(* IEC 61131-3 sources: SCLTeamCoder/experiment/datasets/oscat/oscat_code (part 2) *)

(* ---- FACT.st ---- *)
FUNCTION FACT : DINT
VAR_INPUT
    X : INT;
END_VAR
IF X >= 0 AND X <= 12 THEN
	FACT := math.FACTS[X];
ELSE
	FACT := -1;
END_IF;

(* working code without array
IF X > 12 OR X < 0 THEN
	FACT := -1;
ELSIF X < 7 THEN
	FACT := 1;
	FOR i := 2 TO X DO
		FACT := FACT * i;
	END_FOR;
ELSE
	FACT := 5040;
	FOR i := 8 TO X DO
		FACT := FACT * i;
	END_FOR;
END_IF;
*)

(* revision history
hm 4.3.2007		rev 1.1
	changed a critical error where while loop was indefinite.

hm	10.12.2007	rev 1.2
	start value for i has changed to 2 for better performance

hm	10. mar 2008	rev 1.3
	changed output of fact to dint to allow bigger values

hm	27. oct. 2008	rev 1.4
	optimized code

hm	26. mar. 2011	rev 1.5
	using array math.facts
*)
END_FUNCTION

(* ---- FIB.st ---- *)
FUNCTION FIB : DINT
VAR_INPUT
    X : INT;
END_VAR

VAR
    t1 : DINT;
    t2 : DINT;
END_VAR
IF X < 0 OR X > 46 THEN
	FIB := -1;
ELSIF x < 2 THEN
	FIB := X;
	RETURN;
ELSE
	(* the fibonacci number is the sum of the two suceeding fibonaci numbers *)
	(* we store the numbers alternatively in t1 and t2 depending on pt *)
	t2 := 1;
	WHILE X > 3 DO
		X := X-2;
		t1 := t1 + t2;
		t2 := t1 + t2;
	END_WHILE;
	IF X > 2 THEN t1 := t1 + t2; END_IF;
	fib := t1 + t2;
END_IF;

(* alternative code for very big numbers

IF X < 31 THEN
	fib := 0.4472136 * (expn(1.618034,X) - expn(-0.618034,X));
ELSE
	fib := 0.4472133 * expn(1.618034,X);
END_IF;

*)

(* revision history
hm		27. dec 2007	rev 1.0
	original version

hm		2. jan 2008	rev 1.1
	deleted unused variable pt

hm		10. mar 2008	rev 1.2
	changed output to dint instead of real

hm		26. mar. 2008	rev 1.3
	function now returns -1 for input < 0 or > 46

*)
END_FUNCTION

(* ---- FILL.st ---- *)
FUNCTION FILL : string
VAR_INPUT
    C : BYTE;
    L : INT;
END_VAR

VAR
    i : INT;
    sx : STRING[1];
END_VAR
Sx := CHR_TO_STRING(c);
(* limit L to maximum 80 characters the length of a standard string *)
L := LIMIT(0,L,STRING_LENGTH);
(* create a string of characters to be connected to str *)
FOR i := 1 TO 8 DO
	FILL := CONCAT(FILL,FILL);
	IF L.7 THEN FILL := CONCAT(FILL,Sx); END_IF;
	L := SHL(L,1);
END_FOR;

(* revision histroy
hm	29. mar. 2008	rev 1.0
	original release

hm	17. dec. 2008	rev 1.1
	changed function chr to chr_to_string

*)
END_FUNCTION

(* ---- FIND_CHAR.st ---- *)
FUNCTION FIND_CHAR : INT
VAR_INPUT
    str : STRING(STRING_LENGTH);
    pos : INT;
END_VAR

VAR
    i : INT;
    pt : POINTER TO ARRAY [1..255] OF BYTE;
    stop : INT;
    X : BYTE;
END_VAR
pt := ADR(str);
stop := LEN(str);
FOR i := MAX(pos,1) TO stop DO;
	X := pt^[i];
	IF X > 31 AND ((setup.EXTENDED_ASCII AND X <> 127) OR (NOT setup.EXTENDED_ASCII AND X < 127)) THEN
		FIND_CHAR := i;
		RETURN;
	END_IF;
END_FOR;
FIND_CHAR := 0;

(* revision history
hm	29. feb 2008	rev 1.0
	original version

hm	26. mar. 2008	rev 1.1
	char will now accept extended ascii

hm	29. mar. 2008	rev 1.2
	changed STRING to STRING(STRING_LENGTH)

hm	21. oct. 2008	rev 1.3
	changes setup constants
	optimized code
*)
END_FUNCTION

(* ---- FIND_CTRL.st ---- *)
FUNCTION FIND_CTRL : INT
VAR_INPUT
    str : STRING(STRING_LENGTH);
    pos : INT;
END_VAR

VAR
    i : INT;
    pt : POINTER TO ARRAY[1..255] OF BYTE;
    stop : INT;
    x : BYTE;
END_VAR
pt := ADR(str);
stop := LEN(str);
FOR i := MAX(pos,1) TO stop DO;
	x := PT^[I];
	IF x < 32 OR X = 127 THEN
		FIND_CTRL := i;
		RETURN;
	END_IF;
END_FOR;
FIND_CTRL := 0;

(* revision history
hm	29. feb 2008	rev 1.0
	original version

hm	26. mar. 2008	rev 1.1
	character 127 is now recognized as control

hm	29. mar. 2008	rev 1.2
	changed STRING to STRING(STRING_LENGTH)
*)
END_FUNCTION

(* ---- FIND_NONUM.st ---- *)
FUNCTION FIND_NONUM : INT
VAR_INPUT
    str : STRING(STRING_LENGTH);
    pos : INT;
END_VAR

VAR
    i : INT;
    pt : POINTER TO ARRAY[1..255] OF BYTE;
    end : INT;
    X : BYTE;
END_VAR
pt := ADR(str);
end := LEN(str);
FOR i := MAX(pos,1) TO end DO;
	X := pt^[i];
	IF (X < 48 AND X <> 46) OR X > 57 THEN
		FIND_NONUM := i;
		RETURN;
	END_IF;
END_FOR;
FIND_NONUM := 0;

(* revision history
hm	6. oct. 2006	rev 1.0
	original version

hm	29. feb 2008	rev 1.1
	added input pos to start search at position

hm	29. mar. 2008	rev 1.2
	changed STRING to STRING(STRING_LENGTH)

hm	21. oct. 2008	rev 1.3
	optimized code

*)
END_FUNCTION

(* ---- FIND_NUM.st ---- *)
FUNCTION FIND_NUM : INT
VAR_INPUT
    str : STRING(SIZE := STRING_LENGTH);
    pos : INT;
END_VAR

VAR
    i : INT;
    pt : POINTER TO ARRAY[1..255] OF BYTE;
    stop : INT;
    X : BYTE;
END_VAR
pt := ADR(str);
stop := LEN(str);
FOR i := MAX(pos,1) TO stop DO;
	X := pt^[i];
	IF (X > 47 AND X < 58) OR X = 46 THEN
		FIND_NUM := i;
		RETURN;
	END_IF;
END_FOR;
FIND_NUM := 0;

(* revision history
hm	6. oct. 2006	rev 1.0
	original version

hm	29. feb 2008	rev 1.1
	added input pos to start search at position

hm	29. mar. 2008	rev 1.2
	changed STRING to STRING(STRING_LENGTH)

*)
END_FUNCTION

(* ---- FINDB.st ---- *)
FUNCTION FINDB : INT
VAR_INPUT
    str1 : STRING(STRING_LENGTH);
    str2 : STRING(STRING_LENGTH);
END_VAR

VAR
    pos : INT;
    length : INT;
END_VAR
length := LEN(str2);
FOR pos := LEN(str1) - length + 1 TO 1 BY -1 DO
	IF MID(str1,length,pos) = str2 THEN
		FindB := pos;
		RETURN;
	END_IF;
END_FOR;
FindB := 0;

(* revision history
hm	6. oct 2006		rev 1.0
	original version

hm	15 dec 2007		rev 1.1
	changed code for better performance

hm	29. feb 2008	rev 1.2
	added findb := 0 for compatibility reasons

hm	29. mar. 2008	rev 1.3
	changed STRING to STRING(STRING_LENGTH)
*)
END_FUNCTION

(* ---- FINDB_NONUM.st ---- *)
FUNCTION FINDB_NONUM : INT
VAR_INPUT
    str : STRING(STRING_LENGTH);
END_VAR

VAR
    pos : INT;
    pt : POINTER TO BYTE;
END_VAR
pt := ADR(str) + LEN(str) - 1;
FOR pos := LEN(str) TO 1 BY -1 DO;
	IF (PT^ < 48 AND PT^ <> 46) OR PT^ > 57 THEN
		FINDB_NONUM := pos;
		RETURN;
	END_IF;
	PT := PT - 1;
END_FOR;
FINDB_NONUM := 0;

(* revision history
hm	6. oct 2006		rev 1.0
	original version

hm	29. feb 2008	rev 1.1
	improved performance

hm	29. mar. 2008	rev 1.2
	changed STRING to STRING(STRING_LENGTH)

hm	21. oct. 2008	rev 1.3
	optimized code
*)
END_FUNCTION

(* ---- FINDB_NUM.st ---- *)
FUNCTION FINDB_NUM : INT
VAR_INPUT
    str : STRING:= STRING_LENGTH; // Input variable of type STRING with specified length
END_VAR

VAR
    pos : INT; // Local variable of type INT
    pt : POINTER TO BYTE; // Local variable of type pointer to BYTE
END_VAR
pt := ADR(str) + LEN(str) - 1;
FOR pos := LEN(str) TO 1 BY -1 DO;
	IF (PT^ > 47 AND PT^ < 58) OR PT^ = 46 THEN
		FINDB_NUM := pos;
		RETURN;
	END_IF;
	PT := PT - 1;
END_FOR;
FINDB_NUM := 0;

(* revision history
hm	6. oct 2006		rev 1.0
	original version

hm	29. feb 2008	rev 1.1
	improved performance

hm	29. mar. 2008	rev 1.2
	changed STRING to STRING(STRING_LENGTH)
*)
END_FUNCTION

(* ---- FINDP.st ---- *)
FUNCTION FINDP : INT
VAR_INPUT
    str : STRING[STRING_LENGTH];
    src : STRING[STRING_LENGTH];
    pos : INT;
END_VAR

VAR
    i : INT;
    ls : INT;
    lx : INT;
    stp : INT;
END_VAR
ls := LEN(str);
lx := LEN(src);
IF ls < lx OR lx = 0 THEN RETURN; END_IF;
stp := ls - lx + 1;
FOR i := MAX(pos,1) TO stp DO
	IF MID(str,lx,i) = src THEN
		FINDP := i;
		RETURN;
	END_IF;
END_FOR;
FINDP := 0;

(* revision histroy
hm	4. feb. 2008	rev 1.0
	original release

hm	29. feb 2008	rev 1.1
	ADDED MAX(pos,1) in loop initialization

hm	29. mar. 2008	rev 1.2
	changed STRING to STRING(STRING_LENGTH)
*)
END_FUNCTION

(* ---- FIX.st ---- *)
FUNCTION FIX : string
VAR_INPUT
    str : STRING[STRING_LENGTH];
    L : INT;
    C : BYTE;
    M : INT;
END_VAR

VAR
    N : INT;
    SX : STRING[STRING_LENGTH];
END_VAR
(* make sure L does not exceed the limits of a string *)
N := LIMIT(0,L,STRING_LENGTH) - LEN(str);
IF N <= 0 THEN
	(* truncate the string at length N *)
	IF M = 1 THEN
		FIX := RIGHT(str,L);
	ELSE
		FIX := LEFT(str,L);
	END_IF;
ELSIF M = 1 THEN
	(* connect fill characters at the beginning *)
	sx := FILL(C,N);
	FIX := CONCAT(sx,str);
ELSIF M = 2 THEN
	(* center str beween fill characters *)
	(* for an uneven number of fill characters, there is one more at the end *)
	sx := FILL(C,SHR(N+1,1));
	FIX := CONCAT(str,sx);
	SX := LEFT(sx,SHR(N,1));
	FIX := CONCAT(sx,FIX);
ELSE
	(* connect fill characters at the end *)
	SX := FILL(C,N);
	FIX := CONCAT(str,SX);
END_IF;

(* revision histroy
hm	29. mar. 2008	rev 1.0
	original release

*)
END_FUNCTION

(* ---- FLOAT_TO_REAL.st ---- *)
FUNCTION FLOAT_TO_REAL : REAL
VAR_INPUT
    FLT : STRING[20];
END_VAR

VAR
    pt : POINTER TO ARRAY[1..20] OF BYTE;
    i : INT;
    X : BYTE;
    sign : INT := 1;
    stop : INT;
    tmp : DINT;
    d : INT;
END_VAR
pt := ADR(FLT);
stop := LEN(FLT);

(* we first check for sign and exit if first number or dot is reached *)
FOR i := 1 TO stop DO
	X := pt^[i];
	IF X > 47 AND X < 58 OR X = 46 THEN
		EXIT;
	ELSIF X = 45 THEN
		(* code 45 is sign *)
		sign := -1;
	END_IF;
END_FOR;

(* now we scan numbers till end or dot or E is reached *)
FOR i := i TO stop DO
	X := pt^[i];
	IF X = 44 OR X = 46 OR X = 69 OR X = 101 THEN
		EXIT;
	(* calculate the value of the digit *)
	ELSIF X > 47 AND x < 58 THEN
		tmp := tmp * 10 + X - 48;
	END_IF;
END_FOR;

(* process the portion after the comma if comma or dot is reached exit if exponent starts *)
IF x = 44 OR X = 46 THEN
	FOR i := i + 1 TO stop DO
		X := pt^[i];
		IF X = 69 OR X = 101 THEN
			EXIT;
		ELSIF x > 47 AND x < 58 THEN
			tmp := tmp * 10 + X - 48;
			d := d - 1;
		END_IF;
	END_FOR;
END_IF;

(* process exponent if present *)
IF X = 69 OR X = 101 THEN
	d := d + DEC_TO_INT(RIGHT(FLT, stop - i));
END_IF;

FLOAT_TO_REAL :=  EXPN(10, d) * DINT_TO_REAL(TMP * SIGN);

(* revision histroy
hm	22. jun. 2008	rev 1.0
	original release

hm	2. oct. 2008	rev 1.1
	fixed an error, characters 8 and 9 would not be converted

hm	22. oct. 2008	rev 1.2
	last fix was not done correctly

hm	23. oct. 2008	rev 1.3
	optimzed code
*)
END_FUNCTION

(* ---- FLOOR.st ---- *)
FUNCTION FLOOR : INT
VAR_INPUT
    X : REAL;
END_VAR
FLOOR := REAL_TO_INT(X);
IF FLOOR > X THEN
	FLOOR := FLOOR - 1;
END_IF;

(* revision history
hm		7. feb 2007		rev 1.0
	originlal version

hm		21. mar. 2008	rev 1.1
	replaced trunc with real_to_int for compatibility reasons

*)
END_FUNCTION

(* ---- FLOOR2.st ---- *)
FUNCTION FLOOR2 : DINT
VAR_INPUT
    X : REAL;
END_VAR
FLOOR2 := REAL_TO_DINT(X);
IF DINT_TO_REAL(FLOOR2) > X THEN
	FLOOR2 := FLOOR2 - 1;
END_IF;

(* revision history
hm	21. mar. 2008	rev 1.0
	originlal version

hm	4. apr. 2008	rev 1.1
	added type conversion to avoid warnings under codesys 3.0
*)
END_FUNCTION

(* ---- FRACT.st ---- *)
FUNCTION FRACT : REAL
VAR_INPUT
    x : REAL;
END_VAR
IF ABS(x) < 2.0E9 THEN
	FRACT := x - DINT_TO_REAL(D_TRUNC(x));
ELSE
	FRACT := 0.0;
END_IF;

(* revision history
hm	4. aug 2006	rev 1.0
	original version

hm	11. mar 2008	rev 1.1
	added dint_to_real for compatibility reasons
	now returns 0 for number > 2e9
	changed input to x

hm	21. mar. 2008	rev 1.2
	use D_trunc instead of TRUNC for compatibility reasons

hm	10. mar. 2009	rev 1.3
	real constants updated to new systax using dot

*)
END_FUNCTION

(* ---- FRMP_B.st ---- *)
FUNCTION FRMP_B : BYTE
VAR_INPUT
    START : BYTE;
    DIR   : BOOL;
    TD    : TIME;
    TR    : TIME;
END_VAR
IF TD < TR THEN
	FRMP_B := MIN(DWORD_TO_BYTE(SHL(TIME_TO_DWORD(TD), 8) / TIME_TO_DWORD(TR)), SEL(DIR, START, BYTE#255 - START));
	IF DIR THEN
		FRMP_B := START + FRMP_B;
	ELSE
		FRMP_B := START - FRMP_B;
	END_IF;
ELSE
	FRMP_B := SEL(DIR, 0, 255);
END_IF;

(* revision history

17. feb. 2011	rev 1.0
	new module

*)
END_FUNCTION

(* ---- FSTRING_TO_BYTE.st ---- *)
FUNCTION FSTRING_TO_BYTE : BYTE
VAR_INPUT
    IN: STRING[12];
END_VAR
IF LEFT(IN, 2) = '2#' THEN
	(* we need to convert binary *)
	FSTRING_TO_BYTE := BIN_TO_BYTE(RIGHT(in, LEN(in) - 2));
ELSIF LEFT(in, 2) = '8#' THEN
	(* weneed to convert octals *)
	FSTRING_TO_BYTE := OCT_TO_BYTE(RIGHT(in, LEN(in) - 2));
ELSIF LEFT(in, 3) = '16#' THEN
	(* we need to convert hexadecimal *)
	FSTRING_TO_BYTE := HEX_TO_BYTE(RIGHT(in, LEN(in) - 3));
ELSE
	(* we assume decimal representation *)
	FSTRING_TO_BYTE := DEC_TO_BYTE(CLEAN(in,'0123456789'));
END_IF;

(* revision histroy
hm	18. jun. 2008	rev 1.0
	original release

hm	20. sep. 2008	rev 1.1
	changed length of input string from 20 to 12
*)
END_FUNCTION

(* ---- FSTRING_TO_DT.st ---- *)
FUNCTION FSTRING_TO_DT : DT
VAR_INPUT
    SDT: STRING[60];    // Input variable for source data text
    FMT: STRING[60];    // Input variable for format
END_VAR

VAR CONSTANT
    ignore: STRING[1] := '*';  // ignore character is *
    fchar: STRING[1] := '#';    // format character is #
END_VAR

VAR
    c: STRING[1];    // local variable for character
    tmp: STRING[20];  // local variable for temporary storage
    end: INT;         // local variable for end indicator
    dy: INT := 1970;  // local variable for year, initialized to 1970
    dm: INT := 1;     // local variable for month, initialized to 1
    dd: INT := 1;     // local variable for day, initialized to 1
    th: INT;         // local variable for hour
    tm: INT;         // local variable for minute
    ts: INT;         // local variable for second
END_VAR
(* scan input string *)
WHILE fmt <> '' DO
	c := LEFT(fmt,1);
	IF c = ignore THEN
		(* skip ignore characters *)
		fmt := DELETE(fmt,1,1);
		sdt := DELETE(sdt,1,1);
	ELSIF C = fchar THEN
		(* format chracter found skip format char and read identifier *)
		(* store format identifier in c and skip to next char in fmt *)
		c := MID(fmt,1,2);
		fmt := DELETE(fmt,2,1);
		(* extract the substring until the end of sdt or to next char of fmt *)
		IF fmt = '' THEN
			tmp := sdt;
		ELSE
			(* serach for end of substring *)
			end := FIND(sdt, LEFT(fmt,1))-1;
			tmp := LEFT(sdt, end);
			sdt := DELETE(sdt, end,1);
		END_IF;
		(* extract information from substring *)
		IF c = 'Y' THEN
			dy := STRING_TO_INT(tmp);
			IF dy < 100 THEN dy := dy + 2000; END_IF;
		ELSIF c = 'M' THEN
			dm := STRING_TO_INT(tmp);
		ELSIF c = 'N' THEN
			dm := FSTRING_TO_MONTH(tmp,0);
		ELSIF c = 'D' THEN
			dd := STRING_TO_INT(tmp);
		ELSIF c = 'h' THEN
			th := STRING_TO_INT(tmp);
		ELSIF c = 'm' THEN
			tm := STRING_TO_INT(tmp);
		ELSIF c = 's' THEN
			ts := STRING_TO_INT(tmp);
		END_IF;
	ELSIF c = LEFT(sdt,1) THEN
		(* skip matching characters *)
		fmt := DELETE(fmt,1,1);
		sdt := DELETE(sdt,1,1);
	ELSE
		RETURN;
	END_IF;
END_WHILE;

FSTRING_TO_DT := SET_DT(dy,dm,dd,th,tm,ts);

(* revision histroy
hm	24. sep. 2008	rev 1.0
	original release

*)
END_FUNCTION

(* ---- FSTRING_TO_DWORD.st ---- *)
FUNCTION FSTRING_TO_DWORD : DWORD
VAR_INPUT
    IN : STRING[40];
END_VAR
IF LEFT(IN, 2) = '2#' THEN
	(* we need to convert binary *)
	FSTRING_TO_DWORD := BIN_TO_DWORD(RIGHT(in, LEN(in) - 2));
ELSIF LEFT(in, 2) = '8#' THEN
	(* weneed to convert octals *)
	FSTRING_TO_DWORD := OCT_TO_DWORD(RIGHT(in, LEN(in) - 2));
ELSIF LEFT(in, 3) = '16#' THEN
	(* we need to convert hexadecimal *)
	FSTRING_TO_DWORD := HEX_TO_DWORD(RIGHT(in, LEN(in) - 3));
ELSE
	(* we assume decimal representation *)
	FSTRING_TO_DWORD := DEC_TO_DWORD(CLEAN(in,'0123456789'));
END_IF;

(* revision histroy
hm	18. jun. 2008	rev 1.0
	original release

hm	20. sep. 2008	rev 1.1
	changed length of input dtring from 20 to 40

*)
END_FUNCTION

(* ---- FSTRING_TO_MONTH.st ---- *)
FUNCTION FSTRING_TO_MONTH : INT
VAR_INPUT
    MTH : STRING(20);
    LANG : INT;
END_VAR

VAR
    lx : INT;
END_VAR
IF LANG = 0 THEN lx := LANGUAGE.DEFAULT; ELSE lx := MIN(LANG, LANGUAGE.LMAX); END_IF;
MTH := TRIM(mth);
MTH := CAPITALIZE(LOWERCASE(MTH));

FOR FSTRING_TO_MONTH := 1 TO 12 DO
	IF MTH = language.MONTHS[lx, FSTRING_TO_MONTH] THEN RETURN; END_IF;
	IF MTH = language.MONTHS3[lx, FSTRING_TO_MONTH] THEN RETURN; END_IF;
END_FOR;

(* since no name matched try to decode as integer *)
FSTRING_TO_MONTH := STRING_TO_INT(MTH);

(* revision histroy
hm	25. sep. 2008	rev 1.0
	original release

hm	19. oct. 2008	rev 1.1
	changed language setup constants

hm	25. oct. 2008	rev 1.2
	optimized code
*)
END_FUNCTION

(* ---- FSTRING_TO_WEEK.st ---- *)
FUNCTION FSTRING_TO_WEEK : BYTE
VAR_INPUT
    WEEK : STRING[60];
    LANG : INT;
END_VAR

VAR
    pos : INT;
END_VAR
pos := FIND(WEEK, ',');
WHILE pos > 0 DO
	FSTRING_TO_WEEK := FSTRING_TO_WEEK OR SHR(BYTE#128, FSTRING_TO_WEEKDAY(MID(WEEK, pos - 1, 1), LANG));
	WEEK := RIGHT(WEEK, LEN(Week) - pos);
	pos := FIND(WEEK, ',');
END_WHILE;
FSTRING_TO_WEEK := (FSTRING_TO_WEEK OR SHR(BYTE#128, FSTRING_TO_WEEKDAY(WEEK, LANG))) AND BYTE#127;

(* revision histroy
hm	18. jun. 2008	rev 1.0
	original release

hm	25. oct. 2008	rev 1.1
	using language defauls and input lang
*)
END_FUNCTION

(* ---- FSTRING_TO_WEEKDAY.st ---- *)
FUNCTION FSTRING_TO_WEEKDAY : INT
VAR_INPUT
    WDAY : STRING[20];
    LANG : INT;
END_VAR

VAR
    tmp : STRING[2];
    i : INT;
    ly : INT;
END_VAR
IF LANG = 0 THEN ly := LANGUAGE.DEFAULT; ELSE ly := MIN(LANG, LANGUAGE.LMAX); END_IF;
(* tmp needs to be calculated first otherwise find can return wrong values *)
tmp := TRIM(wday);
tmp := CAPITALIZE(LOWERCASE(tmp));
FOR i := 1 TO 7 DO
	IF language.WEEKDAYS2[ly, i] = tmp THEN
		FSTRING_TO_WEEKDAY := i;
		RETURN;
	END_IF;
END_FOR;
FSTRING_TO_WEEKDAY := STRING_TO_INT(WDAY);

(* revision histroy
hm	18. jun. 2008	rev 1.0
	original release

hm	18. jul. 2008	rev 1.1
	changed nested call of left(trim()) for compatibility reasons

hm	25. oct. 2008	rev 1.2
	using language constants
*)
END_FUNCTION

(* ---- GAMMA.st ---- *)
FUNCTION GAMMA : REAL
VAR_INPUT
    X : REAL;
END_VAR
IF x > 0.0 THEN
	GAMMA := SQRT(math.PI2 / X) * EXPT(math.E_INV * (x + 1.0 / (12.0 * x - 0.1 / X)), X);
END_IF;

(* the stirling formula is not very accurate for small values of X
IF X >=0 THEN GAMMA := SQRT(math.PI2 * X) * EXPT(X / math.E, X); END_IF;
*)

(* revision history
hm	10.12.2007	rev 1.0
	original version

hm	18. oct. 2008	rev 1.1
	using math constants

hm	26. oct. 2008	rev 1.2
	using new formula with better accuracy

hm	10. mar. 2009	rev 1.3
	real constants updated to new systax using dot

*)
END_FUNCTION

(* ---- GAUSS.st ---- *)
FUNCTION GAUSS : REAL
VAR_INPUT
    X : REAL;
    U : REAL;
    SI : REAL;
END_VAR

VAR
    temp : REAL;
    si_inv : REAL;
END_VAR
temp := X - U;
si_inv := 1.0  / si;
GAUSS := EXP(Temp * Temp * si_inv * si_inv * - 0.5) * 0.39894228 * si_inv;

(* revision hisdtory
hm	6. apr. 2008	rev 1.0
	original version

hm	27. oct. 2008	rev 1.1
	optimized performance

hm	10. mar. 2009	rev 1.2
	real constants updated to new systax using dot

*)
END_FUNCTION

(* ---- GAUSSCD.st ---- *)
FUNCTION GAUSSCD : REAL
VAR_INPUT
    X : REAL;
    U : REAL;
    SI : REAL;
END_VAR
GAUSSCD := (ERF((X - U) / (SI * 1.414213562)) + 1.0) * 0.5;

(* revision hisdtory
hm	6. apr. 2008	rev 1.0
	original version

hm	10. mar. 2009	rev 1.1
	real constants updated to new systax using dot

*)
END_FUNCTION

(* ---- GCD.st ---- *)
FUNCTION GCD : INT
VAR_INPUT
    A : DINT;
    B : DINT;
END_VAR

VAR
    t : DINT;
END_VAR
IF A = 0 THEN
	GCD := DINT_TO_INT(ABS(B));
ELSIF B = 0 THEN
	GCD := DINT_TO_INT(ABS(A));
ELSE
	A := ABS(A);
	B := ABS(B);
	GCD := 1;
	WHILE NOT(A.0 OR B.0) DO
		A := SHR(A,1);
		B := SHR(B,1);
		GCD := SHL(GCD,1);
	END_WHILE;
	WHILE A > 0 DO
		IF NOT(A.0) THEN A := SHR(A,1);
		ELSIF NOT(B.0) THEN B := SHR(B,1);
		ELSE
			t:= SHR(ABS(A-B),1);
			IF A < B THEN B := t; ELSE A := T; END_IF;
		END_IF;
	END_WHILE;
	GCD := GCD * DINT_TO_INT(B);
END_IF;

(* revision history
hm	19. jan. 2011	rev 1.0
	original version

*)
END_FUNCTION

(* ---- GDF.st ---- *)
FUNCTION GDF : REAL
VAR_INPUT
    X : REAL;
END_VAR
IF X = 0.0 THEN
	GDF := 0.0;
ELSIF X > 15.0 THEN
	GDF := math.PI05;
ELSIF X < -15.0 THEN
	GDF := -math.PI05;
ELSE
	GDF := ATAN(EXP(X)) * 2.0 - math.PI05;
END_IF;

(* revision history
hm	27. apr. 2008	rev 1.0
	original version

hm	18. oct. 2008	rev 1.1
	using math constants

hm	10. mar. 2009	rev 1.2
	real constants updated to new systax using dot

*)
END_FUNCTION

(* ---- GEO_TO_DEG.st ---- *)
FUNCTION GEO_TO_DEG : REAL
VAR_INPUT
    D : INT;
    M : INT;
    SEC : REAL;
END_VAR
GEO_TO_DEG := INT_TO_REAL(D) + INT_TO_REAL(M) * 0.016666666666667 + sec * 0.00027777777777778;

(* revision histroy
hm	22. jan. 2009	rev 1.0
	original release

*)
END_FUNCTION

(* ---- GOLD.st ---- *)
FUNCTION GOLD : REAL
VAR_INPUT
    X : REAL;
END_VAR
GOLD := (X + SQRT(X*X + 4.0)) * 0.5;

(* revision history
hm	27. apr. 2008	rev 1.0
	original version

hm	10. mar. 2009	rev 1.1
	real constants updated to new systax using dot

*)
END_FUNCTION

(* ---- GRAY_TO_BYTE.st ---- *)
FUNCTION GRAY_TO_BYTE : BYTE
VAR_INPUT
    IN : BYTE;
END_VAR
GRAY_TO_BYTE := SHR(IN,4) XOR IN;
GRAY_TO_BYTE := SHR(GRAY_TO_BYTE,2) XOR GRAY_TO_BYTE;
GRAY_TO_BYTE := SHR(GRAY_TO_BYTE,1) XOR GRAY_TO_BYTE;

(* revision history
hm	9. nov. 2009	rev 1.0
	original version

*)
END_FUNCTION

(* ---- HEX_TO_BYTE.st ---- *)
FUNCTION HEX_TO_BYTE : BYTE
VAR_INPUT
    HEX : STRING(5);
END_VAR

VAR
    pt : POINTER TO BYTE;
    i : INT;
    X : BYTE;
    stop : INT;
END_VAR
pt := ADR(hex);
stop := LEN(hex);
FOR I := 1 TO stop DO
	(* read the first character and subtract 48 to get value in decimal 0 = 48 *)
	x := pt^;
	(* calculate the value of the digit *)
	IF X > 47 AND x < 58 THEN
		HEX_TO_BYTE := SHL(HEX_TO_BYTE,4) + X - 48;
	ELSIF X > 64 AND X < 71 THEN
		HEX_TO_BYTE := SHL(HEX_TO_BYTE,4) + X - 55;
	ELSIF X > 96 AND X < 103 THEN
		HEX_TO_BYTE := SHL(HEX_TO_BYTE,4) + X - 87;
	END_IF;
	pt := pt + 1;
END_FOR;

(* revision histroy
hm	18. jun. 2008	rev 1.0
	original release

hm	20. sep.2008	rev 1.1
	changed length of input string from 20 to 5

*)
END_FUNCTION

(* ---- HEX_TO_DWORD.st ---- *)
FUNCTION HEX_TO_DWORD : DWORD
VAR_INPUT
    Hex: STRING[20];
END_VAR

VAR
    pt: POINTER TO BYTE;
    i: INT;
    X: BYTE;
    stop: INT;
END_VAR
pt := ADR(hex);
stop := LEN(hex);
FOR I := 1 TO stop DO
	(* read the first character and subtract 48 to get value in decimal 0 = 48 *)
	x := pt^;
	(* calculate the value of the digit *)
	IF X > 47 AND x < 58 THEN
		HEX_TO_DWORD := SHL(HEX_TO_DWORD,4) + X - 48;
	ELSIF X > 64 AND X < 71 THEN
		HEX_TO_DWORD := SHL(HEX_TO_DWORD,4) + X - 55;
	ELSIF X > 96 AND X < 103 THEN
		HEX_TO_DWORD := SHL(HEX_TO_DWORD,4) + X - 87;
	END_IF;
	pt := pt + 1;
END_FOR;

(* revision histroy
hm	2.10.2007		rev 1.0
	original release

hm	19.11.2007		rev 1.1
	changed type of function from int to dword

hm 	4. mar 2008		rev 1.2
	added support for a..f and return 0 for invalid string

hm	29. mar. 2008	rev 1.3
	changed STRING to STRING(8)

hm	18. jun. 2008	rev 1.4
	changed input hex to STRING(20)
	function now ignores wrong characters
*)
END_FUNCTION

(* ---- HOUR.st ---- *)
FUNCTION HOUR : INT
VAR_INPUT
    itod : TIME_OF_DAY; // Declaration of input variable itod of type TIME_OF_DAY
END_VAR
HOUR := DWORD_TO_INT(TOD_TO_DWORD(itod) / 3600000);

(* change history
hm 4. aug 2006	rev 1.0
	original version

hm 2.10.2006 	rev 1.1
	changed name of input to itod

*)
END_FUNCTION

(* ---- HOUR_OF_DT.st ---- *)
FUNCTION HOUR_OF_DT : INT
VAR_INPUT
    XDT : DT;
END_VAR
HOUR_OF_DT := DWORD_TO_INT((DT_TO_DWORD(XDT) MOD 86400) / 3600);

(* revision history
hm		6.9.2008	rev 1.0
	original version

*)
END_FUNCTION

(* ---- HOUR_TO_TIME.st ---- *)
FUNCTION HOUR_TO_TIME : TIME
VAR_INPUT
    IN : REAL;
END_VAR
HOUR_TO_TIME := DWORD_TO_TIME(REAL_TO_DWORD(IN * 3600000));

(* revision history
hm		4. aug 2006	rev 1.0
	original version

hm	14. mar. 2008	rev 1.1
	rounded the input after the last digit

hm	24. feb. 2009	rev 1.2
	changed input to IN
*)
END_FUNCTION

(* ---- HOUR_TO_TOD.st ---- *)
FUNCTION HOUR_TO_TOD : TOD
VAR_INPUT
    IN : REAL;
END_VAR
HOUR_TO_TOD := DWORD_TO_TOD(REAL_TO_DWORD(IN * 3600000));

(* revision history
hm	4. aug. 2006	rev 1.0
	original version

hm	14. mar. 2008	rev 1.1
	rounded the input after the last digit

hm	24. feb. 2009	rev 1.2
	changed input to IN
*)
END_FUNCTION

(* ---- HYPOT.st ---- *)
FUNCTION HYPOT : REAL
VAR_INPUT
    X : REAL;
    Y : REAL;
END_VAR
HYPOT := SQRT(x*x + y*y);

(* revision history
hm	21. feb 2008	rev 1.0
	original version

*)
END_FUNCTION

(* ---- INC.st ---- *)
FUNCTION INC : INT
VAR_INPUT
    X : INT;
    D : INT;
    M : INT;
END_VAR
INC := (X + D + M + 1) MOD (M + 1);

(* revision history
hm	7. feb 2007		REV 1.0
	original version

hm	15. jan 2008	rev 1.1
	allow for neagtive increment

*)
END_FUNCTION

(* ---- INC1.st ---- *)
FUNCTION INC1 : INT
VAR_INPUT
    X : INT;
    N : INT;
END_VAR
IF X >= N - 1 THEN
	INC1 := 0;
ELSE
	INC1 := X + 1;
END_IF;

(* revision history
hm	13. oct. 2008	rev 1.0
	original version

hm	22. oct. 2008	rev 1.1
	added statement to return value for compatibility reasons

hm	23. feb. 2009	rev 1.2
 	when inc1 is called with X >= N inc will continue with 0
*)
END_FUNCTION

(* ---- INC2.st ---- *)
FUNCTION INC2 : INT
VAR_INPUT
    X : INT;
    D : INT;
    L : INT;
    U : INT;
END_VAR

VAR
    tmp : INT;
END_VAR
tmp := U - L + 1;
INC2 := (X + D - L + tmp) MOD tmp + L;

(* revision history
hm	29. jun. 2008		REV 1.0
	original version

*)
END_FUNCTION

(* ---- INT_TO_BCDC.st ---- *)
FUNCTION INT_TO_BCDC : BYTE
VAR_INPUT
    IN : INT;
END_VAR
INT_TO_BCDC := SHL(INT_TO_BYTE(IN / INT#10),4) OR INT_TO_BYTE(in MOD INT#10);

(* revision history
hm	13.12.2007
	original version

hm	30.6.2008	rev 1.1
	changed name INT_TO_BCD to INT_TO_BCDC to avoid collision with util.lib
	corrected error in code

*)
END_FUNCTION

(* ---- INV.st ---- *)
FUNCTION INV : REAL
VAR_INPUT
    X : REAL;
END_VAR
IF X <> 0.0 THEN INV := 1.0 / X; END_IF;

(* revision history
hm	26. oct. 2008	rev 1.0
	original version

hm	10. mar. 2009	rev 1.1
	real constants updated to new systax using dot

*)
END_FUNCTION

(* ---- IS_ALNUM.st ---- *)
FUNCTION IS_ALNUM : BOOL
VAR_INPUT
    str : STRING(STRING_LENGTH);
END_VAR_INPUT

VAR
    L : INT;
    pt : POINTER TO BYTE;
    pos : INT;
END_VAR
PT := ADR(str);
L := LEN(str);
FOR pos := 1 TO L DO
	IF NOT (ISC_ALPHA(pt^) OR ISC_NUM(pt^)) THEN
		IS_ALNUM := FALSE;
		RETURN;
	END_IF;
    	PT := PT + 1;
END_FOR;
IS_ALNUM := L > 0;

(* revision history
hm	29. feb 2008	rev 1.0
	original version

hm	29. mar. 2008	rev 1.1
	changed STRING to STRING(STRING_LENGTH)
*)
END_FUNCTION

(* ---- IS_ALPHA.st ---- *)
FUNCTION IS_ALPHA : BOOL
VAR_INPUT
    str: STRING(STRING_LENGTH);
END_VAR

VAR
    L: INT;
    pt: POINTER TO BYTE;
    pos: INT;
END_VAR
PT := ADR(str);
L := LEN(str);
FOR pos := 1 TO L DO
	IF NOT ISC_ALPHA(pt^) THEN
		IS_ALPHA := FALSE;
		RETURN;
	END_IF;
    	PT := PT + 1;
END_FOR;
IS_ALPHA := L > 0;

(* revision history
hm	29. feb 2008	rev 1.0
	original version

hm	29. mar. 2008	rev 1.1
	changed STRING to STRING(STRING_LENGTH)
*)
END_FUNCTION

(* ---- IS_CC.st ---- *)
FUNCTION IS_CC : BOOL
VAR_INPUT
    str : STRING(STRING_LENGTH);
    cmp : STRING(STRING_LENGTH);
END_VAR

VAR
    L : INT;
    pos : INT;
END_VAR
L := LEN(str);
FOR pos := 1 TO L DO
	IF FIND(CMP,MID(str,1,pos)) = 0 THEN RETURN; END_IF;
END_FOR;
IS_CC := L > 0;

(* revision history
hm	19. mar 2008	rev 1.0
	original version

hm	29. mar. 2008	rev 1.1
	changed STRING to STRING(STRING_LENGTH)
*)
END_FUNCTION

(* ---- IS_CTRL.st ---- *)
FUNCTION IS_CTRL : BOOL
VAR_INPUT
    STR : STRING(STRING_LENGTH);
END_VAR

VAR
    L : INT;
    pt : POINTER TO BYTE;
    pos : INT;
END_VAR
PT := ADR(str);
L := LEN(str);
FOR pos := 1 TO L DO
	IF NOT (ISC_CTRL(pt^)) THEN
		IS_CTRL := FALSE;
		RETURN;
	END_IF;
    	PT := PT + 1;
END_FOR;
IS_CTRL := L > 0;

(* revision history
hm	29. feb. 2008	rev 1.0
	original version

hm	29. mar. 2008	rev 1.1
	changed STRING to STRING(STRING_LENGTH)
*)
END_FUNCTION

(* ---- IS_HEX.st ---- *)
FUNCTION IS_HEX : BOOL
VAR_INPUT
    str : STRING[STRING_LENGTH];
END_VAR

VAR
    L : INT;
    pt : POINTER TO BYTE;
    pos : INT;
END_VAR
PT := ADR(str);
L := LEN(str);
FOR pos := 1 TO L DO
	IF NOT (ISC_HEX(pt^)) THEN
		IS_HEX := FALSE;
		RETURN;
	END_IF;
    	PT := PT + 1;
END_FOR;
IS_HEX := L > 0;

(* revision history
hm	29. feb 2008	rev 1.0
	original version

hm	29. mar. 2008	rev 1.1
	changed STRING to STRING(STRING_LENGTH)
*)
END_FUNCTION

(* ---- IS_LOWER.st ---- *)
FUNCTION IS_LOWER : BOOL
VAR_INPUT
    str : STRING[STRING_LENGTH]; // Input variable declaration
END_VAR

VAR
    l : INT; // Local variable declaration
    pt : POINTER TO BYTE; // Pointer variable declaration
    pos : INT; // Position variable declaration
END_VAR
PT := ADR(str);
L := LEN(str);
FOR pos := 1 TO L DO
	IF NOT (ISC_LOWER(pt^)) THEN
		IS_LOWER := FALSE;
		RETURN;
	END_IF;
    	PT := PT + 1;
END_FOR;
IS_LOWER := L > 0;

(* revision history
hm	29. feb 2008	rev 1.0
	original version

hm	29. mar. 2008	rev 1.1
	changed STRING to STRING(STRING_LENGTH)
*)
END_FUNCTION

(* ---- IS_NCC.st ---- *)
FUNCTION IS_NCC : BOOL
VAR_INPUT
    str : STRING[STRING_LENGTH];
    cmp : STRING[STRING_LENGTH];
END_VAR

VAR
    L : INT;
    pos : INT;
END_VAR
L := LEN(str);
FOR pos := 1 TO L DO
	IF FIND(CMP,MID(str,1,pos)) > 0 THEN RETURN; END_IF;
END_FOR;
IS_NCC := TRUE;

(* revision history
hm	19. mar 2008	rev 1.0
	original version

hm	29. mar. 2008	rev 1.1
	changed STRING to STRING(STRING_LENGTH)
*)
END_FUNCTION

(* ---- IS_NUM.st ---- *)
FUNCTION IS_NUM : BOOL
VAR_INPUT
    str : STRING[STRING_LENGTH];  // Input variable of type STRING with specified length
END_VAR

VAR
    L : INT;                       // Local variable of type INT
    pt : POINTER TO BYTE;         // Local variable, pointer to BYTE
    pos : INT;                    // Local variable of type INT
END_VAR
PT := ADR(str);
L := LEN(str);
FOR pos := 1 TO L DO
	IF NOT (ISC_NUM(pt^)) THEN
		IS_NUM := FALSE;
		RETURN;
	END_IF;
    	PT := PT + 1;
END_FOR;
IS_NUM := L > 0;

(* revision history
hm	29. feb 2008	rev 1.0
	original version

hm	29. mar. 2008	rev 1.1
	changed STRING to STRING(STRING_LENGTH)
*)
END_FUNCTION

(* ---- IS_SORTED.st ---- *)
FUNCTION IS_SORTED : BOOL
VAR_INPUT
    pt : ^ ARRAY [0..32000] OF REAL; // Pointer to an array of REAL
    size : UINT; // Size variable of type UINT
END_VAR

VAR
    stop : INT; // Local variable of type INT
    i : INT; // Local variable of type INT
END_VAR
stop := UINT_TO_INT(SHR(size,2)-2);
FOR i := 0 TO stop DO
	IF pt^[i] > pt^[i+1] THEN
		IS_SORTED := FALSE;
		RETURN;
	END_IF;
END_FOR;

IS_SORTED := TRUE;

(* revision history

hm 	29. mar. 2008 	rev 1.0
	original version

hm	4. apr. 2008	rev 1.1
	added type conversion to avoid warnings under codesys 3.0
*)
END_FUNCTION

(* ---- IS_UPPER.st ---- *)
FUNCTION IS_UPPER : BOOL
VAR_INPUT
    str : STRING; // Length to be defined as per application requirements
END_VAR

VAR
    L : INT;
    pt : POINTER TO BYTE;
    pos : INT;
END_VAR
PT := ADR(str);
L := LEN(str);
FOR pos := 1 TO L DO
	IF NOT (ISC_UPPER(pt^)) THEN
		IS_UPPER := FALSE;
		RETURN;
	END_IF;
    	PT := PT + 1;
END_FOR;
IS_UPPER := L > 0;

(* revision history
hm	29. feb 2008	rev 1.0
	original version

hm	29. mar. 2008	rev 1.1
	changed STRING to STRING(STRING_LENGTH)
*)
END_FUNCTION

(* ---- ISC_ALPHA.st ---- *)
FUNCTION ISC_ALPHA : BOOL
#VAR_INPUT
    IN : BYTE;
END_VAR
IF setup.EXTENDED_ASCII THEN
	ISC_ALPHA := (in > 64 AND in < 91) OR (in > 191  AND in <> 215 AND in <> 247) OR (in > 96 AND in < 123);
ELSE
	ISC_ALPHA := (IN > 64 AND IN < 91) OR (in > 96 AND in < 123);
END_IF;

(* revision history
hm	6. mar. 2008	rev 1.0
	original version

hm	19. oct. 2008	rev 1.1
	changes setup constants
*)
END_FUNCTION

(* ---- ISC_CTRL.st ---- *)
FUNCTION ISC_CTRL : BOOL
VAR_INPUT
    IN : BYTE;
END_VAR
ISC_CTRL := IN < 32 OR IN = 127;

(* revision history
hm		6. mar. 2008	rev 1.0
	original version

*)
END_FUNCTION

(* ---- ISC_HEX.st ---- *)
FUNCTION ISC_HEX : BOOL
VAR_INPUT
    IN : BYTE;
END_VAR
ISC_HEX := (IN > 47 AND IN < 58) OR (IN > 64 AND IN < 71) OR (IN > 96 AND IN < 103);

(* revision history
hm		6. mar. 2008	rev 1.0
	original version

*)
END_FUNCTION

(* ---- ISC_LOWER.st ---- *)
FUNCTION ISC_LOWER : BOOL
VAR_INPUT
    IN : BYTE; // Input variable
END_VAR
IF setup.EXTENDED_ASCII THEN
	ISC_LOWER := ((in > 96) AND (in < 123)) OR ((in > 222) AND (in <> 247));
ELSE
	ISC_LOWER := ((in > 96) AND (in < 123));
END_IF;

(* revision history
hm	6. mar. 2008	rev 1.0
	original version

hm	19. oct. 2008	rev 1.1
	changes setup constants
*)
END_FUNCTION

(* ---- ISC_NUM.st ---- *)
FUNCTION ISC_NUM : BOOL
VAR_INPUT
    IN : BYTE;
END_VAR
ISC_NUM := IN > 47 AND IN < 58;

(* revision history
hm		6. mar. 2008	rev 1.0
	original version

*)
END_FUNCTION

(* ---- ISC_UPPER.st ---- *)
FUNCTION ISC_UPPER : BOOL
VAR_INPUT
    IN : BYTE;
END_VAR
IF setup.EXTENDED_ASCII THEN
	ISC_UPPER :=  ((in > 64) AND (in < 91)) OR (((in > 191) AND (in < 223)) AND (in <> 215));
ELSE
	ISC_UPPER := ((in > 64) AND (in < 91));
END_IF;

(* revision history
hm	6. mar. 2008	rev 1.0
	original version

hm	19. oct. 2008	rev 1.1
	changes setup constants

*)
END_FUNCTION

(* ---- JD2000.st ---- *)
FUNCTION JD2000 : REAL
VAR_INPUT
    DTI : TIME;
END_VAR
JD2000 := DWORD_TO_REAL(DT_TO_DWORD(DTI) - 946728000) / 86400.0;

(* revision histroy
hm	15. jul. 2008	rev 1.0
	original release

*)
END_FUNCTION

(* ---- K_TO_C.st ---- *)
FUNCTION K_TO_C : REAL
VAR_INPUT
    Kelvin : REAL;
END_VAR
K_TO_C := Kelvin + phys.T0;

(* revision history

hm	4. aug 2006	rev 1.0
	original version

hm	19. aug 2009	rev 1.1
	fixed calculation error

*)
END_FUNCTION

(* ---- KMH_TO_MS.st ---- *)
FUNCTION KMH_TO_MS : REAL
VAR_INPUT
    kmh : REAL;
END_VAR
KMH_TO_MS := kmh * 0.2777777777777;

(* revision history
hm	4. feb 2007		rev 1.0
	original version

hm	6. jan 2008		rev 1.1
	improved performance

*)
END_FUNCTION

(* ---- LAMBERT_W.st ---- *)
FUNCTION LAMBERT_W : REAL
VAR_INPUT
    X : REAL;
END_VAR

VAR
    w : REAL;
    i : INT;
    we : REAL;
    w1e : REAL;
    last : DWORD;
    ewx : REAL;
END_VAR
(* check for valid input and return -1000 if too low *)
IF x < -0.367879441171442 THEN
	LAMBERT_W := -1000.0;
	RETURN;
(* return 0 if x = 0 *)
ELSIF x = 0.0 THEN
	RETURN;
(* first an estimate is calculated *)
ELSIF x <= 500.0 THEN
	w := LN(x + 1.0);
	w := 0.665 * (1.0 + 0.0195 * w) * w + 0.04;
ELSE
	w := LN(x - 4.0) - (1.0 - 1.0/LN(x)) * LN(LN(x));
END_IF;
(* use estimate to calculate exact result *)
FOR i := 0 TO 5 DO
	ewx := EXP(w);
	we := w * ewx - x;
	w1e := (w+1.0) * ewx;
	last := REAL_TO_DW(w) AND 16#FFFF_FFFC;
	w := w - (we / (w1e - (w+2.0) * we / (2.0 * w + 2.0)));
	IF (REAL_TO_DW(w) AND 16#FFFF_FFFC) = last THEN EXIT; END_IF;
END_FOR;
LAMBERT_W := w;

(* revision hisdtory
hm	26. oct. 2008	rev 1.0
	original version

hm	10. mar. 2009	rev 1.1
	real constants updated to new systax using dot

*)
END_FUNCTION

(* ---- LANGEVIN.st ---- *)
FUNCTION LANGEVIN : REAL
VAR_INPUT
    X : REAL;
END_VAR
IF X = 0.0 THEN
	LANGEVIN := 0.0;
ELSE
	LANGEVIN := COTH(X) - 1.0 / X;
END_IF;

(* revision history
hm	10.12.2007	rev 1.0
	original version

hm	11. mar 2008	rev 1.1
	changed formula to avoid problems when x = 0

hm	10. mar. 2009	rev 1.2
	real constants updated to new systax using dot

*)
END_FUNCTION

(* ---- LEAP_DAY.st ---- *)
FUNCTION LEAP_DAY : BOOL
VAR_INPUT
    IDATE : DATE;
END_VAR
LEAP_DAY := DATE_TO_UDINT(IDATE) MOD 126230400 = 68169600;

(* change history

hm 	15. jun. 2008	rev 1.0
	original version

hm	7. oct. 2008	rev 1.1
	changed function month to month_of_date

hm	24. jan. 2011	rev 1.2
	improved performance
*)
END_FUNCTION

(* ---- LEAP_OF_DATE.st ---- *)
FUNCTION LEAP_OF_DATE : BOOL
VAR_INPUT
    idate: DATE;
END_VAR
LEAP_OF_DATE := SHL(((DATE_TO_DWORD(idate) + 43200) / 31557600), 30) = 16#80000000;

(* change history

2.10.2006		rev 1.1
the function now calls leap_year to accomodate further accuracy.
the function now works for any year from 1970 to 2100

8. jan 2008		rev 1.2
	improved code for better performance

28. jan. 2011	rev 1.3
	improved performance
*)
END_FUNCTION

(* ---- LEAP_YEAR.st ---- *)
FUNCTION LEAP_YEAR : BOOL
VAR_INPUT
    yr : INT;  // Variable for year
END_VAR
LEAP_YEAR := SHL(yr,14) = 0;

(* this code was used prior to rev 1.1

IF yr MOD 400 = 0 THEN leap_year := TRUE;
ELSIF yr MOD 100 = 0 THEN leap_year := FALSE;
ELSIF yr MOD 4 =0 THEN leap_year := TRUE;
ELSE leap_year := FALSE;
END_IF;

*)

(* change history

hm 	2.10.2006		rev 1.1
	the function now works for any year from 1970 up to 2100

hm	1. oct 2007		rev 1.2
	chaged code for higher performance
*)
END_FUNCTION

(* ---- LINEAR_INT.st ---- *)
FUNCTION LINEAR_INT : REAL
VAR_INPUT
    X : REAL;
    XY : ARRAY[1..20, 0..1] OF REAL;
    Pts : INT;
END_VAR

VAR
    i : INT;
END_VAR
(*make sure n is bound within the array size *)
pts := MIN(pts,20);

(* calculate the linear segement interpolation *)
i := 2;
(* search for segment and calculate output
	below and above the defined segments we interpolate the last segment *)
WHILE (i < pts) AND (XY[i,0] < X) DO
	i := i + 1;
END_WHILE;

(* calculate the output value on the corresponding segment coordinates *)
LINEAR_INT := ((XY[i,1] - XY[i-1,1]) * X - XY[i,1] * XY[i-1,0] + XY[i-1,1] * XY[i,0]) / (XY[i,0] - XY[i-1,0]);

(* revision history
hm	7. oct 2007		rev 1.0
	original version

hm	27 dec 2007		rev 1.1
	changed code for better performance
*)
END_FUNCTION

(* ---- LIST_ADD.st ---- *)
FUNCTION LIST_ADD : BOOL
VAR_INPUT
    SEP : BYTE;
    INS : STRING(LIST_LENGTH);
END_VAR

VAR_IN_OUT
    LIST : STRING(LIST_LENGTH);
END_VAR

VAR
    sx : STRING(1);
END_VAR
sx := CHR_TO_STRING(SEP);			(* convert separation character to string *)
INS := CONCAT(sx, INS);					(* start element with separation character *)

IF LEN(LIST) + LEN(INS) > LIST_LENGTH THEN
	LIST_ADD := FALSE;					(* return false if element does not fit *)
ELSE
	LIST := CONCAT(LIST, INS);
	LIST_ADD := TRUE;
END_IF;

(* revision histroy

hm	21. mar. 2011	rev 2.0
	original release
*)
END_FUNCTION

(* ---- LIST_CLEAN.st ---- *)
FUNCTION LIST_CLEAN : BOOL
VAR_INPUT
    SEP : BYTE;
END_VAR

VAR_IN_OUT
    LIST : STRING[LIST_LENGTH];
END_VAR

VAR
    pt : POINTER TO ARRAY[1..LIST_LENGTH] OF BYTE;
    read : INT := 1;
    write : INT := 1;
    last : BYTE;
    c : BYTE;
END_VAR
pt := ADR(LIST);

FOR read := 1 TO LIST_LENGTH DO
	c := pt^[read];								(* read character from list *)
	IF c = 0 THEN EXIT;						(* exit the loop if character definbes end of string *)
	ELSIF c <> SEP OR sep <> last THEN	(* copy element from read to write position unless a double sep character is present *)
		pt^[write] := c;
		write := write + 1;
	END_IF;
	last := c;									(* remember last character *)
END_FOR;

IF last = SEP THEN write := write - 1; END_IF;		(* if last character is sep then delete empty element at end *)
IF write <= STRING_LENGTH THEN pt^[write] := 0;	 END_IF;		(* terminate string with 0 *)

LIST_CLEAN := TRUE;						(* retrun TRUE *)

(* revision histroy
hm	28. jun. 2008	rev 1.0
	original release

hm	19. jan. 2011	rev 1.1
	changed string(255) to string(LIST_LENGTH)

hm	21. mar. 2011	rev 2.0
	all elements start with SEP

*)
END_FUNCTION

(* ---- LIST_GET.st ---- *)
FUNCTION LIST_GET : string
VAR_INPUT
    SEP : BYTE;       // Input variable
    POS : INT;        // Input variable
END_VAR

VAR_IN_OUT
    LIST : STRING(LIST_LENGTH);  // InOut variable
END_VAR

VAR
    i : INT := 1;      // Local variable with initial value
    o : INT := 1;      // Local variable with initial value
    pt : POINTER TO ARRAY[1..LIST_LENGTH] OF BYTE; // Pointer to array of BYTE
    po : POINTER TO ARRAY[1..LIST_LENGTH] OF BYTE; // Pointer to array of BYTE
    cnt : INT := 0;    // Local variable with initial value
    c : BYTE;          // Local variable
END_VAR
pt := ADR(LIST);							(* load pointers *)
po := ADR(LIST_GET);

REPEAT
	c := pt^[i];
	IF cnt = pos THEN						(* copy element to output string *)
		IF c = SEP  THEN EXIT; END_IF;		(* next element stop copy and finish *)
		po^[o] := c;
		o := o + 1;
	ELSIF c = SEP THEN
		cnt := cnt + 1;
	END_IF;
	i := i + 1;
UNTIL
	(i = LIST_LENGTH) OR (c = 0)
END_REPEAT;
po^[o] := 0;						(* close the output string *)

(* revision histroy
hm	20. jun. 2008	rev 1.0
	original release

hm	19. jan. 2011	rev 1.1
	changed string(255) to strring(LIST_LENGTH)

hm	21. mar. 2011	rev 2.0
	all list elements start with SEP
*)
END_FUNCTION

(* ---- LIST_INSERT.st ---- *)
FUNCTION LIST_INSERT : BOOL
VAR_INPUT
    SEP : BYTE;
    POS : INT;
    INS : STRING(LIST_LENGTH);
END_VAR

VAR_IN_OUT
    LIST : STRING(LIST_LENGTH);
END_VAR

VAR
    pt : POINTER TO ARRAY[1..LIST_LENGTH] OF BYTE;
    read : INT := 1;
    cnt : INT := 1;
    sx : STRING(1);
END_VAR
(* load pointers *)
pt := ADR(LIST);

IF LEN(ins) + 1 + LEN(LIST) > LIST_LENGTH THEN
	LIST_INSERT := FALSE;
ELSE
	LIST_INSERT := TRUE;
	(* search for position *)
	WHILE read < LIST_LENGTH DO
		IF cnt >= POS THEN
			sx := CHR_TO_STRING(SEP);
			INS := CONCAT(sx, INS);
			LIST := INSERT(LIST, INS, read - 1);
			LIST_INSERT := TRUE;
			RETURN;
		END_IF;
		IF pt^[read]  = 0 THEN				(* list is too short add empty element *)
			pt^[read] := SEP;
			pt^[read + 1] := 0;
		END_IF;
		read := read + 1;
		IF pt^[read] = SEP OR pt^[read] = 0 THEN cnt := cnt + 1; END_IF;
	END_WHILE;
END_IF;

(* revision histroy
hm	28. jun. 2008	rev 1.0
	original release

hm	17. dec. 2008	rev 1.1
	changes name of function chr to chr_to_string

hm	19. jan. 2011	rev 1.2
	changed string(255) to string(LIST_LENGTH)

hm	21. mar. 2011	rev 2.0
	all list elements start with SEP

*)
END_FUNCTION

(* ---- LIST_LEN.st ---- *)
FUNCTION LIST_LEN : INT
VAR_INPUT
    SEP : BYTE;
END_VAR

VAR_IN_OUT
    LIST : STRING(LIST_LENGTH);
END_VAR

VAR
    pt : ^ARRAY[1..LIST_LENGTH] OF BYTE;
    pos : INT := 1;
    c : BYTE;
END_VAR
pt := ADR(LIST);
LIST_LEN := 0;
REPEAT
	c := pt^[pos];
	IF c = SEP THEN LIST_LEN := LIST_LEN + 1; END_IF;
	pos := pos + 1;
UNTIL
	c = 0 OR pos > LIST_LENGTH
END_REPEAT;

(* revision histroy
hm	25. jun. 2008	rev 1.0
	original release

hm	16. oct. 2008	rev 1.1
	fixed a problem where list_len would only work up to LIST_LENGTH

hm	19. jan. 2001	rev 1.2
	changed string(255) to string(LIST_LENGTH)

hm	21. mar. 2011	rev 2.0
	all list elements start with SEP

*)
END_FUNCTION

(* ---- LIST_RETRIEVE.st ---- *)
FUNCTION LIST_RETRIEVE : string
VAR_INPUT
    SEP : BYTE;
    POS : INT;
END_VAR

VAR_IN_OUT
    LIST : STRING(LIST_LENGTH);
END_VAR

VAR
    i : INT;
    o : INT := 1;
    w : INT := 1;
    pt : POINTER TO ARRAY[1..LIST_LENGTH] OF BYTE;
    po : POINTER TO ARRAY[1..LIST_LENGTH] OF BYTE;
    cnt : INT := 0;
    c : BYTE;
END_VAR
(* load pointers *)
pt := ADR(LIST);
po := ADR(LIST_RETRIEVE);

IF pos > 0 THEN
	FOR i := 1 TO LIST_LENGTH DO
		c := pt^[i];
		IF c = 0 THEN
			po^[o] := 0;
			IF cnt < pos THEN pt^[w + 1] := 0; ELSE pt^[w] := 0; END_IF;
			RETURN;
		ELSIF cnt = pos AND c <> SEP THEN				(* we have found the element *)
			po^[o] := pt^[i];
			o := o + 1;
		ELSIF cnt >= pos THEN
			pt^[w] := c;
			w := w + 1;
		ELSE
			w := i;
		END_IF;
		IF c = sep THEN cnt := cnt + 1; END_IF;
	END_FOR;
ELSE
	LIST_RETRIEVE := '';
END_IF;

(* revision histroy
hm	28. jun. 2008	rev 1.0
	original release

hm	19. jan. 2011	rev 1.1
	changed string(255) to string(LIST_LENGTH)

hm	21. mar. 2011	rev 2.0
	all elements start with SEP
*)
END_FUNCTION

(* ---- LIST_RETRIEVE_LAST.st ---- *)
FUNCTION LIST_RETRIEVE_LAST : string
VAR_INPUT
    SEP : BYTE;
END_VAR

VAR_IN_OUT
    LIST : STRING[LENGTH := LIST_LENGTH];
END_VAR

VAR
    i : INT;
    last : INT := 1;
    pt : POINTER TO ARRAY[1..LIST_LENGTH] OF BYTE;
    c : BYTE;
END_VAR
(* load pointers *)
pt := ADR(LIST);

(* search position of last element *)
FOR i := 1 TO LIST_LENGTH DO
	c := pt^[i];
	IF c = 0 THEN
		EXIT;
	ELSIF C = SEP THEN
		last := i;
	END_IF;
END_FOR;
(* return last element of list *)
LIST_RETRIEVE_LAST := MID(LIST, LIST_LENGTH, last + 1);
(* terminate list at i *)
pt^[last] := 0;

(* revision histroy
hm	21. mar. 2011	rev 2.0
	new module
*)
END_FUNCTION

(* ---- LOWERCASE.st ---- *)
FUNCTION LOWERCASE : string
VAR_INPUT
    str: STRING[STRING_LENGTH];
END_VAR

VAR
    PT: POINTER TO BYTE;
    pos: INT;
    l: INT;
END_VAR
PT := ADR(LOWERCASE);
lowercase := str;
l := LEN(str);
FOR pos := 1 TO l DO
	pt^ := TO_LOWER(pt^);
	PT := PT + 1;
END_FOR;

(* revision histroy
hm	6. oct. 2006	rev 1.0
	original release

hm	4. feb. 2008	rev 1.1
	improved performance
	added Ä.Ö,Ü

hm	6. mar. 2008	rev 1.2
	added support for exteded Ascii

hm	29. mar. 2008	rev 1.3
	changed STRING to STRING(STRING_LENGTH)
*)
END_FUNCTION

(* ---- LTIME_TO_UTC.st ---- *)
FUNCTION LTIME_TO_UTC : DT
VAR_INPUT
    LOCAL_TIME : DT;
    DST : BOOL;
    TIME_ZONE_OFFSET : INT;
END_VAR
LTIME_TO_UTC := UDINT_TO_DT(DT_TO_UDINT(LOCAL_TIME) - INT_TO_UDINT(TIME_ZONE_OFFSET) * 60);
IF DST THEN LTIME_TO_UTC := LTIME_TO_UTC - T#1h; END_IF;

(* revision history
hm 5.7.2007		rev 1.0
	original version

hm 5.11.2007		rev 1.1
	replaced literal constant with variable because of error in möller ecp4 compiler

hm	12.nov 2007	rev 1.2
	changed Type of time_zone_offset from time to int to allow for time zones with negative offset

hm	8. dec 2007	rev 1.3
	corrected a problem with time_zone_offset

hm	14. oct. 2008	rev 1.4
	changed time_zone_offset from int to real to allow for half hour offset

hm	20. oct. 2006	rev 1.5
	changed time_zone_offset from Real to INT, now in Minutes

hm	27. feb. 2009	rev 1.6
	added type conversions to avoid warnings under codesys 3.0

ks	13. nov. 2009	rev 1.7
	corrected error in formula

*)
END_FUNCTION

(* ---- MANUAL.st ---- *)
FUNCTION MANUAL : BOOL
VAR_INPUT
    IN : BOOL;
    ON : BOOL;
    OFF : BOOL;
END_VAR
MANUAL := NOT OFF AND (IN OR ON);

(* revision history
hm	21. nov 2008	rev 1.0
	original version

*)
END_FUNCTION

(* ---- MAX3.st ---- *)
FUNCTION MAX3 : REAL
VAR_INPUT
    in1 : REAL;
    in2 : REAL;
    in3 : REAL;
END_VAR
MAX3 := MAX(MAX(IN1,IN2),IN3);

(* revision history
hm	1.1.2007	rev 1.0
	original release

hm	18. mar. 2011	rev 1.1
	improve performance

*)
END_FUNCTION

(* ---- MID3.st ---- *)
FUNCTION MID3 : REAL
VAR_INPUT
    IN1 : REAL;
    IN2 : REAL;
    IN3 : REAL;
END_VAR
IF IN1 > IN2 THEN MID3 := IN1; IN1 := IN2; IN2 := MID3; END_IF;
IF IN2 > IN3 THEN IN2 := IN3; END_IF;
MID3 := SEL(IN1 > IN2, IN2, IN1);

(*
hm	1.1.2007	rev 1.1
	rewrote the function for better performance

hm	18. mar. 2011	rev 1.2
	improve performance
*)
END_FUNCTION

(* ---- MIN3.st ---- *)
FUNCTION MIN3 : REAL
VAR_INPUT
    in1 : REAL;
    in2 : REAL;
    in3 : REAL;
END_VAR
MIN3 := MIN(MIN(IN1,IN2),IN3);

(* revision history
hm	1.1.2007	rev 1.0
	original release

hm	18. mar. 2011	rev 1.1
	improve performance

*)
END_FUNCTION

(* ---- MINUTE.st ---- *)
FUNCTION MINUTE : INT
VAR_INPUT
    itod : TOD;
END_VAR
MINUTE := DWORD_TO_INT(TOD_TO_DWORD(itod) / 60000 - TOD_TO_DWORD(itod) / 3600000 * 60);

(* change history

2.10.2006 changes name of input to itod

*)
END_FUNCTION

(* ---- MINUTE_OF_DT.st ---- *)
FUNCTION MINUTE_OF_DT : INT
VAR_INPUT
    XDT : DT;
END_VAR
MINUTE_OF_DT := DWORD_TO_INT(DT_TO_DWORD(XDT) MOD 3600) / 60;

(* revision history
hm		6.9.2008	rev 1.0
	original version

*)
END_FUNCTION

(* ---- MINUTE_TO_TIME.st ---- *)
FUNCTION MINUTE_TO_TIME : TIME
VAR_INPUT
    IN : REAL;
END_VAR
MINUTE_TO_TIME := DWORD_TO_TIME(REAL_TO_DWORD(IN * 60000.0));

(* revision history
hm	4. aug 2006	rev 1.0
	original version

hm	14. mar 2008	rev 1.1
	rounded the input after the last digit

hm	24. feb. 2009	rev 1.2
	changed input to IN

*)
END_FUNCTION

(* ---- MIRROR.st ---- *)
FUNCTION MIRROR : string
VAR_INPUT
    str: STRING(STRING_LENGTH);
END_VAR

VAR
    pi: POINTER TO ARRAY[1..255] OF BYTE;
    po: POINTER TO BYTE;
    lx: INT;
    i: INT;
END_VAR
pi := ADR(str);
po := ADR(mirror);
lx := LEN(str);
FOR i := lx TO 1 BY - 1 DO
	po^ := pi^[i];
	po := po + 1;
END_FOR;
(* close output string *)
po^:= 0;

(* revision histroy
hm	4. feb. 2008	rev 1.0
	original release

hm	29. mar. 2008	rev 1.1
	changed STRING to STRING(STRING_LENGTH)
*)
END_FUNCTION

(* ---- MIX.st ---- *)
FUNCTION MIX : REAL
VAR_INPUT
    A : REAL;
    B : REAL;
    M : REAL;
END_VAR
MIX := (1.0 - M) * A + M * B;

(* revision history
hm	19. Nov 2007	rev 1.0
	original version

hm	10. mar 2009	rev 1.1
	real constants updated to new systax using dot

*)
END_FUNCTION

(* ---- MODR.st ---- *)
FUNCTION MODR : REAL
VAR_INPUT
    IN : REAL;
    DIVI : REAL;
END_VAR
IF divi = 0.0 THEN
	MODR := 0.0;
ELSE
	MODR := in - DINT_TO_REAL(FLOOR2(in / divi)) * divi;
END_IF;

(* revision history

hm	4. aug.2006		rev 1.0

hm	28. jan.2007	rev 1.1
	modr(x,0) will deliver the result 0

hm	21. mar 2008	rev 1.2
	use D_trunc for compatibility reasons

hm	4. apr. 2008	rev 1.3
	added type conversion to avoid warnings under codesys 3.0

hm	31. oct. 2008	rev 1.4
	changed algorithm to the more common version using floor instead of TRUNC

hm	10. mar. 2009	rev 1.5
	real constants updated to new systax using dot

*)
END_FUNCTION

(* ---- MONTH_BEGIN.st ---- *)
FUNCTION MONTH_BEGIN : DATE
VAR_INPUT
    idate : DATE;
END_VAR
MONTH_BEGIN := DWORD_TO_DATE(DATE_TO_DWORD(idate) - INT_TO_DWORD(DAY_OF_MONTH(idate) - 1) * 86400);

(* revision history
hm	15. jun. 2008	rev 1.0
	original version

*)
END_FUNCTION

(* ---- MONTH_END.st ---- *)
FUNCTION MONTH_END : DATE
VAR_INPUT
    IDATE : DATE;
END_VAR
MONTH_END := DWORD_TO_DATE(DATE_TO_DWORD(SET_DATE(YEAR_OF_DATE(idate),MONTH_OF_DATE(idate)+1,1)) - 86400);

(* revision history
hm	15. jun. 2008	rev 1.0
	original version

hm	7. oct. 2008	rev 1.1
	changed function year to year_of_date
	changed function month to month_of_date

*)
END_FUNCTION

(* ---- MONTH_OF_DATE.st ---- *)
FUNCTION MONTH_OF_DATE : INT
VAR_INPUT
    IDATE: DATE;
END_VAR
MONTH_OF_DATE := DAY_OF_YEAR(idate);
IF MONTH_OF_DATE < 32 THEN
	MONTH_OF_DATE := 1;
ELSIF LEAP_OF_DATE(IDATE) THEN
	MONTH_OF_DATE := (MONTH_OF_DATE * 53 + 1668) / 1623;
ELSE
	MONTH_OF_DATE := (MONTH_OF_DATE * 53 + 1700) / 1620;
END_IF;

(* code for rev 1.2
MONTH_OF_DATE := DAY_OF_YEAR(IDATE);
IF LEAP_OF_DATE(IDATE) THEN
	CASE MONTH_OF_DATE OF
		1..31 	:	MONTH_OF_DATE := 1;
		32..60	:	MONTH_OF_DATE := 2;
		61..91	:	MONTH_OF_DATE := 3;
		92..121 :	MONTH_OF_DATE := 4;
		122..152:	MONTH_OF_DATE := 5;
		153..182:	MONTH_OF_DATE := 6;
		183..213:	MONTH_OF_DATE := 7;
		214..244:	MONTH_OF_DATE := 8;
		245..274:	MONTH_OF_DATE := 9;
		275..305:	MONTH_OF_DATE := 10;
		306..335:	MONTH_OF_DATE := 11;
		336..366:	MONTH_OF_DATE := 12;
	END_CASE;
ELSE
	CASE MONTH_OF_DATE OF
		1..31 	:	MONTH_OF_DATE := 1;
		32..59	:	MONTH_OF_DATE := 2;
		60..90	:	MONTH_OF_DATE := 3;
		91..120 :	MONTH_OF_DATE := 4;
		121..151:	MONTH_OF_DATE := 5;
		152..181:	MONTH_OF_DATE := 6;
		182..212:	MONTH_OF_DATE := 7;
		213..243:	MONTH_OF_DATE := 8;
		244..273:	MONTH_OF_DATE := 9;
		274..304:	MONTH_OF_DATE := 10;
		305..334:	MONTH_OF_DATE := 11;
		335..365:	MONTH_OF_DATE := 12;
	END_CASE;
END_IF;
*)

(* revision history
hm	1. aug 2006	rev 1.0
	original version

hm	1. okt 2007	rev 1.1
	replaced old code (string conversion) with mathematics
	the execution time is now multiple times faster.

hm	7. oct. 2008	rev 1.2
	changed name of function from month to MONTH_OF_DATE

hm	27. mar. 2009	rev 1.3
	new improved code

*)
END_FUNCTION

(* ---- MONTH_TO_STRING.st ---- *)
FUNCTION MONTH_TO_STRING : string
VAR_INPUT
    MTH : INT;
    LANG : INT;
    LX : INT;
END_VAR

VAR
    ly : INT;
END_VAR
IF LANG <= 0 THEN Ly := LANGUAGE.DEFAULT; ELSE ly := MIN(LANG, language.LMAX); END_IF;
IF MTH < 1 OR MTH > 12 THEN
	RETURN;
ELSIF LX = 0 THEN
	MONTH_TO_STRING := language.MONTHS[ly, MTH];
ELSIF Lx = 3 THEN
	MONTH_TO_STRING := language.MONTHS3[ly, MTH];
END_IF;

(* revisison history

hm	21. sep. 2008	rev 1.0
	original version

hm	19. oct. 2008	rev 1.1
	changed language setup constants

hm 16.  jul 2024   rev 1.2
       addaed boundary check to respect array limits
*)
END_FUNCTION

(* ---- MS_TO_BFT.st ---- *)
FUNCTION MS_TO_BFT : INT
VAR_INPUT
    MS : REAL;
END_VAR
MS_TO_BFT := REAL_TO_INT(EXPT(MS * 1.196172, 0.666667));

(* revision history
hm	12. 6. 2008		rev 1.0
	original version

*)
END_FUNCTION

(* ---- MS_TO_KMH.st ---- *)
FUNCTION MS_TO_KMH : REAL
VAR_INPUT
    ms : REAL;
END_VAR
MS_TO_KMH := ms * 3.6;
END_FUNCTION

(* ---- MUL_ADD.st ---- *)
FUNCTION MUL_ADD : REAL
VAR_INPUT
    X : REAL;
    K : REAL;
    O : REAL;
END_VAR
MUL_ADD := X * K + O;

(* revision history
hm	28. feb 2007
	original version

hm	11.nov 2007		rev 1.1
	deleted preset values for K and O this makes no sense for a function

*)
END_FUNCTION

(* ---- MULTI_IN.st ---- *)
FUNCTION MULTI_IN : REAL
VAR_INPUT
    in_1 : REAL;
    in_2 : REAL;
    in_3 : REAL;
    default : REAL;
    in_min : REAL;
    in_max : REAL;
    mode : BYTE;
END_VAR

VAR
    count : INT;
    F1 : BOOL;
    F2 : BOOL;
    F3 : BOOL;
END_VAR
F1 :=  in_1 > in_min AND in_1 < in_max;
F2 :=  in_2 > in_min AND in_2 < in_max;
F3 :=  in_3 > in_min AND in_3 < in_max;

CASE mode OF
0:	count := 0;
	IF F1 THEN
		count := count + 1;
		MULTI_IN := in_1;
	ELSE
		MULTI_IN := 0.0;
	END_IF;
	IF F2 THEN
		count := count + 1;
		MULTI_IN := MULTI_IN + in_2;
	END_IF;
	IF F3 THEN
		count := count + 1;
		MULTI_IN := MULTI_IN + in_3;
	END_IF;
	MULTI_IN := SEL(count = 0, MULTI_IN / INT_TO_REAL(count), default);

1:	MULTI_IN := SEL(F1, default, IN_1);

2:	MULTI_IN := SEL(F2, default, IN_2);

3:	MULTI_IN := SEL(F3, default, IN_3);

4:	MULTI_IN := default;

5:	MULTI_IN := SEL(F1, in_max, IN_1);
	IF F2 AND in_2 < MULTI_IN THEN MULTI_IN := in_2; END_IF;
	IF F3 AND in_3 < MULTI_IN THEN MULTI_IN := in_3; END_IF;
	IF MULTI_IN = in_max THEN MULTI_IN := default; END_IF;

6:	MULTI_IN := SEL(F1, in_min, IN_1);
	IF F2 AND in_2 > MULTI_IN THEN MULTI_IN := in_2; END_IF;
	IF F3 AND in_3 > MULTI_IN THEN MULTI_IN := in_3; END_IF;
	IF MULTI_IN = in_min THEN MULTI_IN := default; END_IF;

7:	IF F1 AND F2 AND F3 THEN MULTI_IN := MID3(in_1, in_2, in_3);
	ELSIF F1 AND F2 THEN MULTI_IN := MIN(in_1, in_2);
	ELSIF F1 AND F3 THEN MULTI_IN := MIN(in_1, in_3);
	ELSIF F2 AND F3 THEN MULTI_IN := MIN(in_2, in_3);
	ELSIF F1 THEN MULTI_IN := in_1;
	ELSIF F2 THEN MULTI_IN := in_2;
	ELSIF F3 THEN MULTI_IN := in_3;
	ELSE MULTI_IN := default;
	END_IF;

END_CASE;

(*
hm 1.1.2007		rev 1.1
	changed midr to mid3 function

hm	14. 10. 2008	rev 1.2
	corrected an error for in_3 overrange detection
	improved performance

hm	11. mar. 2009	rev 1.3
	changed real constants to use dot syntax

hm	18. jul. 2009	rev 1.4
	improved performance
*)
END_FUNCTION

(* ---- MULTIME.st ---- *)
FUNCTION MULTIME : TIME
VAR_INPUT
    t : TIME;
    M : REAL;
END_VAR
MULTIME := DWORD_TO_TIME(REAL_TO_DWORD(DWORD_TO_REAL(TIME_TO_DWORD(t))*M));

(* revision history
hm		2. oct 2006	rev 1.0
	original version

hm		14. mar 2008	rev 1.1
	rounded the result after the last digit

*)
END_FUNCTION

(* ---- MUX_2.st ---- *)
FUNCTION MUX_2 : BOOL
VAR_INPUT
    D0 : BOOL;
    D1 : BOOL;
    A0 : BOOL;
END_VAR
MUX_2 := SEL(A0, D0, D1);

(*
revision history:
hm	5.10.2006		rev 1.1
	changed to ST Langage for better portability.

hm	16. oct. 2008	rev 1.2
	improved performance

*)
END_FUNCTION

(* ---- MUX_4.st ---- *)
FUNCTION MUX_4 : BOOL
VAR_INPUT
    D0 : BOOL;
    D1 : BOOL;
    D2 : BOOL;
    D3 : BOOL;
    A0 : BOOL;
    A1 : BOOL;
END_VAR
IF A1 THEN
	MUX_4 := SEL(A0, D2, D3);
ELSE
	MUX_4 := SEL(A0, D0, D1);
END_IF;

(*
revision history:
hm 	5.10.2006		rev 1.1
	rewritten to ST for better portability

hm	16. oct. 2008	rev 1.2
	improved performance

*)
END_FUNCTION

(* ---- MUX_R2.st ---- *)
FUNCTION MUX_R2 : REAL
VAR_INPUT
    IN0 : REAL;
    IN1 : REAL;
    A : BOOL;
END_VAR
MUX_R2 := SEL(A, IN0, IN1);

(* revision history
hm	19. jan. 2007	rev 1.0
	original version

hm	16. oct. 2008	rev 1.1
	improved performance

*)
END_FUNCTION

(* ---- MUX_R4.st ---- *)
FUNCTION MUX_R4 : REAL
VAR_INPUT
    IN0 : REAL;
    IN1 : REAL;
    IN2 : REAL;
    IN3 : REAL;
    A0 : BOOL;
    A1 : BOOL;
END_VAR
IF A1 THEN
	MUX_R4 := SEL(A0, IN2, IN3);
ELSE
	MUX_R4 := SEL(A0, IN0, IN1);
END_IF;

(* revision history
hm	19. jan 2007	rev 1.0
	original version

hm	16. oct. 2008	rev 1.1
	improved performance
*)
END_FUNCTION

(* ---- NEGX.st ---- *)
FUNCTION NEGX : REAL
VAR_INPUT
    X : REAL;
END_VAR
NEGX := -X;

(* revision history
hm	26. oct. 2008	rev 1.0
	original version

*)
END_FUNCTION

(* ---- OCT_TO_BYTE.st ---- *)
FUNCTION OCT_TO_BYTE : BYTE
VAR_INPUT
    OCT : STRING[10];
END_VAR

VAR
    pt : POINTER TO BYTE;
    i : INT;
    X : BYTE;
    stop : INT;
END_VAR
pt := ADR(oct);
stop := LEN(oct);
FOR I := 1 TO stop DO
	(* read the first character and subtract 48 to get value in decimal 0 = 48 *)
	x := pt^;
	(* calculate the value of the digit *)
	IF X > 47 AND x < 56 THEN
		OCT_TO_BYTE := SHL(OCT_TO_BYTE,3) + X - 48;
	END_IF;
	pt := pt + 1;
END_FOR;

(* revision histroy
hm	18. jun. 2008	rev 1.0
	original release

hm	20. sep. 2008	rev 1.1
	changed length of input string from 20 to 10

*)
END_FUNCTION

(* ---- OCT_TO_DWORD.st ---- *)
FUNCTION OCT_TO_DWORD : DWORD
VAR_INPUT
    OCT : STRING[20];
END_VAR

VAR
    pt : POINTER TO BYTE;
    i : INT;
    X : BYTE;
    stop : INT;
END_VAR
pt := ADR(oct);
stop := LEN(oct);
FOR I := 1 TO stop DO
	(* read the first character and subtract 48 to get value in decimal 0 = 48 *)
	x := pt^;
	(* calculate the value of the digit *)
	IF X > 47 AND x < 56 THEN
		OCT_TO_DWORD := SHL(OCT_TO_DWORD,3) + X - 48;
	END_IF;
	pt := pt + 1;
END_FOR;

(* revision histroy
hm	18. jun. 2008	rev 1.0
	original release

*)
END_FUNCTION

(* ---- OFFSET.st ---- *)
FUNCTION OFFSET : REAL
VAR_INPUT
    X : REAL;
    O1 : BOOL;
    O2 : BOOL;
    O3 : BOOL;
    O4 : BOOL;
    D : BOOL;
    Offset_1 : REAL;
    Offset_2 : REAL;
    Offset_3 : REAL;
    Offset_4 : REAL;
    default : REAL;
END_VAR
IF D THEN OFFSET := default; ELSE OFFSET := X; END_IF;
IF O1 THEN OFFSET := OFFSET + offset_1; END_IF;
IF O2 THEN OFFSET := OFFSET + offset_2; END_IF;
IF O3 THEN OFFSET := OFFSET + offset_3; END_IF;
IF O4 THEN OFFSET := OFFSET + offset_4; END_IF;

(* revision history
hm	12. jan 2007
	original version

*)
END_FUNCTION

(* ---- OFFSET2.st ---- *)
FUNCTION OFFSET2 : REAL
VAR_INPUT
    X : REAL;
    O1 : BOOL;
    O2 : BOOL;
    O3 : BOOL;
    O4 : BOOL;
    D : BOOL;
    Offset_1 : REAL;
    Offset_2 : REAL;
    Offset_3 : REAL;
    Offset_4 : REAL;
    default : REAL;
END_VAR
IF D THEN OFFSET2 := default; ELSE OFFSET2 := X; END_IF;
IF O4 THEN OFFSET2 := OFFSET2 + offset_4;
ELSIF O3 THEN OFFSET2 := OFFSET2 + offset_3;
ELSIF O2 THEN OFFSET2 := OFFSET2 + offset_2;
ELSIF O1 THEN OFFSET2 := OFFSET2 + offset_1;
END_IF;
END_FUNCTION

(* ---- OM_TO_F.st ---- *)
FUNCTION OM_TO_F : REAL
VAR_INPUT
    OM : REAL;
END_VAR
OM_TO_F := OM / math.PI2;

(* revision history
hm	22. jan. 2007	rev 1.0
	original version

hm	18. oct. 2008	rev 1.1
	using math constants

*)
END_FUNCTION

(* ---- OSCAT_VERSION.st ---- *)
FUNCTION OSCAT_VERSION : DWORD
VAR_INPUT
    IN : BOOL;
END_VAR
IF in THEN
	OSCAT_VERSION := DATE_TO_DWORD(D#2024-07-16);
ELSE
	OSCAT_VERSION := 335;
END_IF;

(* revision history
hm	6. oct 2006	rev 1.0
	original version

hm	16. dec 2007	rev 1.1
	added possibility to return date and version depending on IN.

*)
END_FUNCTION

(* ---- OVERRIDE.st ---- *)
FUNCTION OVERRIDE : REAL
VAR_INPUT
    X1 : REAL;
    X2 : REAL;
    X3 : REAL;
    E1 : BOOL;
    E2 : BOOL;
    E3 : BOOL;
END_VAR
IF E1 THEN OVERRIDE := X1; END_IF;
IF E2 AND ABS(x2) > ABS(OVERRIDE) THEN OVERRIDE := X2; END_IF;
IF E3 AND ABS(x3) > ABS(OVERRIDE) THEN OVERRIDE := X3; END_IF;

(* revision history
hm	4.11.2007		rev 1.0
	original version

*)
END_FUNCTION

(* ---- PARITY.st ---- *)
FUNCTION PARITY : BOOL
VAR_INPUT
    in : DWORD;
END_VAR
WHILE in > 0 DO
	PARITY := PARITY XOR in.0 XOR in.1 XOR in.2 XOR in.3;
	in := SHR(in,4);
END_WHILE;

(* code before rev 1.2
WHILE in > 0 DO
	IF in.0 THEN cnt := cnt +1; END_IF;
	in := SHR(in,1);
END_WHILE;
IF (cnt MOD 2) = 1 THEN parity := TRUE; ELSE parity := FALSE; END_IF;
*)

(* revision history

rev 1.0 hm 1 sep 2006
	original version

rev 1.1 hm 10.9.2007
	changed algorithm to improve performance

rev 1.2	hm	8 dec 2007
	changed algorithm to improve performance

rev 1.3	hm	18 feb 2008
	changed algorithm to improve performance
*)
END_FUNCTION

(* ---- PERIOD.st ---- *)
FUNCTION PERIOD : BOOL
VAR_INPUT
    d1: DATE;
    dx: DATE;
    d2: DATE;
END_VAR

VAR
    day1: INT;
    day2: INT;
    dayx: INT;
END_VAR
day1 := DAY_OF_YEAR(d1);
day2 := DAY_OF_YEAR(d2);
dayx := DAY_OF_YEAR(dx);
IF NOT LEAP_OF_DATE(dx) AND dayx > 58 THEN dayx := dayx + 1; END_IF;
IF NOT LEAP_OF_DATE(d1) AND day1 > 58 THEN day1 := day1 + 1; END_IF;
IF NOT LEAP_OF_DATE(d2) AND day2 > 58 THEN day2 := day2 + 1; END_IF;

IF day2 < day1 THEN
	(* the period spans over the new year *)
	PERIOD := dayx <= day2 OR dayx >= day1;
ELSE
	PERIOD := dayx >= day1 AND dayx <= day2;
END_IF;

(* code before rev 1.2
yx := year(dx);
p1 := date_add(d1,0,0,0,yx - year(d1));
p2 := date_add(d2,0,0,0,yx - year(d2));

IF p2 >= p1 THEN
	period := dx <= p2  AND dx >= p1;
ELSE
	period := dx <= p2 OR dx >= p1;
END_IF;
*)

(* revision history

hm		19. sep 2007	rev 1.0
	original version

hm		20. sep 2007	rev 1.1
	corrected a problem with leap year

hm		4. jan 2008		rev 1.2
	changed code for better performance

hm		22. mar. 2008	rev 1.3
	function would deliver wrong results when d1, d2 or dx are a leap_year

*)
END_FUNCTION

(* ---- PERIOD2.st ---- *)
FUNCTION PERIOD2 : BOOL
VAR_INPUT
    DP : ARRAY[0..3, 0..1] OF DATE; // Array of DATEs
    DX : DATE;                     // Single DATE
END_VAR
PERIOD2 := 	(DX >= DP[0,0] AND DX <= DP[0,1]) OR
			(DX >= DP[1,0] AND DX <= DP[1,1]) OR
			(DX >= DP[2,0] AND DX <= DP[2,1]) OR
			(DX >= DP[3,0] AND DX <= DP[3,1]);

(* revision history

hm		27. apr 2008	rev 1.0
	original version

*)
END_FUNCTION

(* ---- POLYNOM_INT.st ---- *)
FUNCTION POLYNOM_INT : REAL
VAR_INPUT
    X : REAL;
    XY : ARRAY[1..5, 0..1] OF REAL;
    Pts : INT;
END_VAR

VAR
    I : INT;
    J : INT;
    stop : INT;
END_VAR
(*make sure n is bound within the array size *)
pts := MIN(pts, 5);

(* this part is only to calculate the polynom parameters, which are then stores in the Y array
	the array values, it is not needed during runtime, unless the parameters will change during runtime
	the remaining code without this setup code can be used within a function to calculate specific functions
	the content of the arrays is then used as constant values within the function *)

FOR i := 1 TO pts DO
	stop := i + 1;
   	FOR j := pts TO stop BY -1 DO
   		XY[j,1] := (XY[j,1] - XY[j-1,1]) / (XY[j,0] - XY[j-i,0]);
	END_FOR;
END_FOR;

(* this part is the actual calculation *)
POLYNOM_INT := 0.0;
FOR i := pts TO 1 BY -1 DO
       POLYNOM_INT := POLYNOM_INT * (X - XY[i,0]) + XY[i,1];
END_FOR;

(* revision history
hm	8. okt 2007	rev 1.0
	original version

hm	17. dec 2007	rev 1.1
	init makes no sense for a function

hm	22. feb 2008	rev 1.2
	improved performance

hm	10. mar. 2009	rev 1.3
	changed syntax of real constants to 0.0

*)
END_FUNCTION

(* ---- PT_TO_F.st ---- *)
FUNCTION PT_TO_F : REAL
VAR_INPUT
    PT : TIME;
END_VAR
PT_TO_F := 1000.0 / DWORD_TO_REAL(TIME_TO_DWORD(PT));

(*	revision history
hm	4. aug. 2006	rev 1.0
	original version

hm	11. mar. 2009	rev 1.1
	real constants updated to new systax using dot

*)
END_FUNCTION

(* ---- R2_ABS.st ---- *)
FUNCTION R2_ABS : REAL2
VAR_INPUT
    X : REAL2;
END_VAR
IF X.RX >= 0.0 THEN
	R2_ABS.RX := X.RX;
	R2_ABS.R1 := X.R1;
ELSE
	R2_ABS.RX := -X.RX;
	R2_ABS.R1 := -X.R1;
END_IF;

(* revision history
hm	21. mar. 2008	rev 1.0
	original version

hm	10. mar. 2009 rev 1.1
	real constants updated to new systax using dot

*)
END_FUNCTION

(* ---- R2_ADD.st ---- *)
FUNCTION R2_ADD : REAL2
VAR_INPUT
    X : Real2;  // Derived type
    Y : REAL;
END_VAR

VAR
    temp : REAL;
END_VAR
temp := X.RX;
R2_ADD.RX := Y + X.R1 + X.RX;
R2_ADD.R1 := temp - R2_ADD.RX + Y + X.R1;

(* revision history
hm		20.3.2008	rev 1.0
	original version

*)
END_FUNCTION

(* ---- R2_ADD2.st ---- *)
FUNCTION R2_ADD2 : REAL2
VAR_INPUT
    X : REAL2;
    Y : REAL2;
END_VAR
R2_ADD2.R1 := X.R1 + Y.R1;
R2_ADD2.RX := X.RX + Y.RX;

(* revision history
hm		20.3.2008	rev 1.0
	original version

*)
END_FUNCTION

(* ---- R2_MUL.st ---- *)
FUNCTION R2_MUL : REAL2
VAR_INPUT
    X : REAL2;
    Y : REAL;
END_VAR
R2_MUL.RX := X.RX * Y;
R2_MUL.R1 := X.R1 * Y;

(* revision history
hm		20.3.2008	rev 1.0
	original version

*)
END_FUNCTION

(* ---- R2_SET.st ---- *)
FUNCTION R2_SET : REAL2
VAR_INPUT
    X : REAL;
END_VAR
R2_SET.RX := X;
R2_SET.R1 := 0.0;

(* revision history
hm	2. jun. 2008	rev 1.0
	original version

hm	10. mar. 2009	rev 1.1
	real constants updated to new systax using dot

*)
END_FUNCTION

(* ---- RAD.st ---- *)
FUNCTION RAD : REAL
VAR_INPUT
    DEG : REAL; // Degrees as input variable
END_VAR
RAD := MODR(0.0174532925199433 * DEG, math.PI2);

(* revision history
hm	4. aug 2006		rev 1.0
	original version

hm 	16. oct 2007	rev 1.1
	added modr statement which prohibits rad to become bigger than 2PI

hm	18. oct 2008	rev 1.2
	using math constants

*)
END_FUNCTION

(* ---- RANGE_TO_BYTE.st ---- *)
FUNCTION RANGE_TO_BYTE : BYTE
VAR_INPUT
    X : REAL;
    low : REAL;
    high : REAL;
END_VAR
RANGE_TO_BYTE := INT_TO_BYTE(DINT_TO_INT(TRUNC((LIMIT(low, X, high) - low) * 255.0 / (high - low))));

(* revision history
hm	9. jan 2008		rev 1.0
	original version

*)
END_FUNCTION

(* ---- RANGE_TO_WORD.st ---- *)
FUNCTION RANGE_TO_WORD : WORD
VAR_INPUT
    X : REAL;
    low : REAL;
    high : REAL;
END_VAR
RANGE_TO_WORD := DINT_TO_WORD(TRUNC((LIMIT(low,X,high)-low) * 65535.0 / (high - low)));

(* revision history
hm	9. jan 2008		rev 1.0
	original version

*)
END_FUNCTION

(* ---- RDM.st ---- *)
FUNCTION RDM : REAL
VAR_INPUT
    last : REAL;
END_VAR

VAR
    tn : DWORD;
    tc : INT;
END_VAR
tn := T_PLC_MS();
tc := BIT_COUNT(tn);
tn.31 := tn.2;
tn.30 := tn.5;
tn.29 := tn.4;
tn.28 := tn.1;
tn.27 := tn.0;
tn.26 := tn.7;
tn.25 := tn.6;
tn.24 := tn.3;
tn := ROL(tn,BIT_COUNT(tn)) OR 16#80000001;
tn := tn MOD 71474513 + INT_TO_DWORD(tc + 77);
RDM := FRACT(DWORD_TO_REAL(tn) / 10000000.0 * (math.E - LIMIT(0.0,last,1.0)));

(*
pt := ADR(temp);
pt^ := (T_PLC_MS() AND 16#007FFFFF) OR 16#3D000000;
RDM := fract(modR(temp*e+pi1, PI1-last) + modR(temp*PI1+e + last,e-last));
*)

(* revision history
hm		16. jan 2007		rev 1.0
	original version

hm		11. nov 2007		rev 1.1
	changed time() into t_plc_ms()

hm		20. nov 2007		rev 1.2
	changed code of temp calculation to avoid overflow in modr due to resuclt would not fit DINT for high timeer values

hm		5. jan 2008		rev 1.3
	changed calculation of temp to avoid problem with high values of t_plc_ms

hm		2. feb 2008		rev 1.4
	changed algorithm to avoind non iec functions and guarantee more randomness

hm	10. mar. 2008		rev 1.5
	make sure last will be between 0 and 1 to avoid invalid results

hm	16. mar. 2008		rev 1.6
	added conversion for tc to avoid warnings under codesys 3.0

hm	18. may. 2008		rev 1.7
	changed constant E to E1

hm	18. oct. 2008		rev 1.8
	using math constants

hm	10. mar. 2009		rev 1.9
	real constants updated to new systax using dot

*)
END_FUNCTION

(* ---- RDM2.st ---- *)
FUNCTION RDM2 : INT
VAR_INPUT
    last : INT;
    low : INT;
    high : INT;
END_VAR
RDM2 := DINT_TO_INT(TRUNC(RDM(FRACT(last * math.PI)) * (high - low + 1)) + low);

(* revision history
hm		29. feb 2008		rev 1.0
	original version

hm		18. oct. 2008		rev 1.1
	using math constants

*)
END_FUNCTION

(* ---- RDMDW.st ---- *)
FUNCTION RDMDW : DWORD
VAR_INPUT
    last: DWORD;
END_VAR

VAR
    RX: REAL;
    M: REAL;
END_VAR
M := BIT_COUNT(last);
RX := RDM(FRACT(M * math.PI));
RDMDW := SHL(REAL_TO_DWORD(rx*65535),16);
RX := RDM(FRACT(M * math.E));
RDMDW := RDMDW OR (REAL_TO_DWORD(rx*65535) AND 16#0000FFFF);

(* revision history
hm		14. mar 2008		rev 1.0
	original version

hm		18. may. 2008		rev 1.1
	changed constant E to E1

hm		18. oct. 2008		rev 1.2
	using math constants

*)
END_FUNCTION

(* ---- REAL_TO_DW.st ---- *)
FUNCTION REAL_TO_DW : DWORD
VAR_INPUT
    X : REAL;  // Input variable of type REAL
END_VAR

VAR
    pt : POINTER TO DWORD;  // Local variable of pointer type to DWORD
END_VAR
pt := ADR(X);
REAL_TO_DW := pt^;

(* revision history
hm	18. apr. 2008
	original version

*)
END_FUNCTION

(* ---- REAL_TO_FRAC.st ---- *)
FUNCTION REAL_TO_FRAC : FRACTION
VAR_INPUT
    X : REAL; // in einen Bruch umzuwandelnder Wert
    N : INT;  // maximale Größe des Nenners
END_VAR

VAR
    temp : DINT; // Merker für Berechnungen
    sign : BOOL; // Vorzeichen vom Eingangswert
    X_gerundet : DINT; // Wert von Bruch, auf ganze Zahl gerundet
    X_ohne_Nachkomma : REAL; // Wert von Bruch, ohne Nachkommastellen
    Numerator : DINT := 1; // Initialwert Zaehler
    Denominator : DINT := 0; // Initialwert Nenner
    Numerator_old : DINT := 0; // Initialwert Zaehler der letzten Berechnung
    Denominator_old : DINT := 1; // Initialwert Nenner der letzten Berechnung
END_VAR
IF X < 0.0 THEN
	sign := TRUE;								(* Vorzeichen merken *)
	X := ABS(X);								(* Absolutwert berechnen *)
END_IF;

REPEAT
	X_gerundet := REAL_TO_DINT(X);

	(* Zaehler berechnen *)
	temp := numerator * X_gerundet + numerator_old;		(* Zaehler um Vorkammawert erweitern *)
	numerator_old := numerator;							(* Zaehler der letzten Berechnung speichern *)
	numerator := temp;									(* Zaehler dieser Berechnung speichern *)

	(* Nenner berechnen *)
	temp := denominator * X_gerundet + denominator_old;	(* Nenner um Vorkammawert erweitern *)
	denominator_old := denominator;						(* Nenner der letzten Berechnung speichern *)
	denominator := temp;								(* Nenner dieser Berechnung speichern *)

	(* Restwert berechnen *)
	X_ohne_Nachkomma := DINT_TO_REAL(X_gerundet);
	IF X = X_ohne_Nachkomma THEN						(* Bruch geht ohne Rest auf *)
		IF ABS(denominator) <= N THEN						(* kein Rundungsfehler *)
			numerator_old := numerator;					(* Numerator_old wird von Funktion zurückgegeben *)
			denominator_old := denominator;			(* Denominator_old wird von Funktion zurückgegeben *)
		END_IF
		EXIT;											(* keine weitere Berechnung notwendig *)
	ELSE
		X := 1.0 / (X - X_ohne_Nachkomma);				(* Kehrwert vom Rest -> Neuer Bruch *)
	END_IF

UNTIL
	ABS(Denominator) > N
END_REPEAT

(* correct sign if X was negative *)
IF sign THEN
	REAL_TO_FRAC.NUMERATOR := -1 * ABS(DINT_TO_INT(numerator_old));
ELSE
	REAL_TO_FRAC.NUMERATOR :=  ABS(DINT_TO_INT(numerator_old));
END_IF
REAL_TO_FRAC.DENOMINATOR := ABS(DINT_TO_INT(denominator_old));

(* revision history
hm		19. jan. 2011	rev 1.0
	original version

ad		06. apr. 2011	rev 1.1
	optimized code
*)
END_FUNCTION

(* ---- REAL_TO_STRF.st ---- *)
FUNCTION REAL_TO_STRF : string
VAR_INPUT
    IN : REAL;
    N : INT;
    D : STRING[1];
END_VAR

VAR
    O : REAL;
    i : INT;
END_VAR
(* LIMIT N to 0 .. 7 *)
N := LIMIT(0,N,7);
(* round the input to N digits and convert to string *)
O := ABS(in) * EXP10(N);
REAL_TO_STRF := DINT_TO_STRING(REAL_TO_DINT(O));
(* add zeroes in front to make sure sting is at least 8 digits long *)
FOR i := LEN(REAL_TO_STRF) TO N DO REAL_TO_STRF := CONCAT('0', REAL_TO_STRF); END_FOR;
(* add a dot if n > 0 *)
IF n > 0 THEN REAL_TO_STRF := INSERT(REAL_TO_STRF, D, LEN(REAL_TO_STRF) - N); END_IF;
(* add a minus sign if in is negative *)
IF in < 0 THEN REAL_TO_STRF := CONCAT('-', REAL_TO_STRF); END_IF;

(* revision history
hm	26 jan 2007	rev 1.0
	original version

hm	20. nov. 2007	rev 1.1
	when N=0 ther will be no dot at the end of the string.

hm	15. dec. 2007	rev 1.2
	changed code for better performance

hm	4. mar. 2008	rev 1.3
	result is now rounded instead of trunc

hm	20. mar. 2008	rev 1.4
	changed trunc to real_to_dint because trunc was generating wrong values on wago 842

hm	29. mar. 2008	rev 1.5
	changed STRING to STRING(20)

hm	4. apr. 2008	rev 1.6
	added variable O to avoid an error uner CoDeSys SP PLCWinNT V2.4

hm	27. feb. 2009	rev 1.7
	added a missing zero for IN < 1

hm 2. jan 2012	rev 1.8
	added input parameter D to specify decimal separator
*)
END_FUNCTION

(* ---- REFLECT.st ---- *)
FUNCTION REFLECT : DWORD
VAR_INPUT
    D : DWORD;
    L : INT;
END_VAR

VAR
    i : INT;
END_VAR
REFLECT := 0;
FOR i := 1 TO L DO
	REFLECT := SHL(REFLECT, 1) OR BOOL_TO_DWORD(D.0);
	D := SHR(D, 1);
END_FOR;
REFLECT := REFLECT OR SHL(D, L);

(* revision history
hm	 16. jan 2011
	new module

*)
END_FUNCTION

(* ---- REFRACTION.st ---- *)
FUNCTION REFRACTION : REAL
VAR_INPUT
    ELEV : REAL;
END_VAR
elev := LIMIT(-1.9, elev, 80.0);
REFRACTION := 0.0174532925199433 / TAN(0.0174532925199433 * (ELEV + 10.3 / (ELEV + 5.11)));

(* revision histroy
hm	14. jul. 2008	rev 1.0
	original release

hm	7. mar. 2009	rev 1.1
	using new formula

*)
END_FUNCTION

(* ---- REPLACE_ALL.st ---- *)
FUNCTION REPLACE_ALL : string
VAR_INPUT
    str : STRING[STRING_LENGTH];
    src : STRING[STRING_LENGTH];
    rep : STRING[STRING_LENGTH];
END_VAR

VAR
    pos : INT;
    lp : INT;
    lx : INT;
END_VAR
REPLACE_ALL := str;
lx := LEN(src);
lp := LEN(rep);
pos := FINDP(REPLACE_ALL, src, 1);
WHILE pos > 0 DO
	REPLACE_ALL := REPLACE(REPLACE_ALL,rep,lx, pos);
	pos := FINDP(REPLACE_ALL, src, pos + lp);
END_WHILE;

(* revision histroy
hm	4. feb. 2008	rev 1.0
	original release

hm	29. mar. 2008	rev 1.1
	changed STRING to STRING(STRING_LENGTH)
*)
END_FUNCTION

(* ---- REPLACE_CHARS.st ---- *)
FUNCTION REPLACE_CHARS : string
VAR_INPUT
    STR : STRING(SIZE := STRING_LENGTH);
    SRC : STRING;
    REP : STRING;
END_VAR

VAR
    a : INT;
    b : INT;
    c : STRING(SIZE := 1);
    stp : INT;
END_VAR
REPLACE_CHARS := STR;
(* make sure rep and src are of same length and length is > 0 *)
a := LEN(src);
b := LEN(rep);
IF a < b THEN
	rep := LEFT(rep, a);
ELSIF b < a THEN
	src := LEFT(src, b);
END_IF;

(* search the string and replace if necessary *)
stp := LEN(str);
FOR a := 1 TO stp DO
	c := MID(REPLACE_CHARS, 1, a);
	b := FIND(src, c);
	IF b > 0 THEN
		REPLACE_CHARS := REPLACE(REPLACE_CHARS, MID(rep, 1, b), 1, a);
	END_IF;
END_FOR;

(* revision history
hm	14. may. 2008	rev 1.0
	original version

*)
END_FUNCTION

(* ---- REPLACE_UML.st ---- *)
FUNCTION REPLACE_UML : string
VAR_INPUT
    str : STRING; // STRING_LENGTH is not defined in XML, use default STRING
END_VAR

VAR
    L : INT;
    pt : POINTER TO BYTE;
    pto : POINTER TO BYTE;
    ptm : POINTER TO BYTE;
    pt1 : POINTER TO BYTE;
    pt2 : POINTER TO BYTE;
    su : STRING[2];
    pos : INT;
END_VAR
PT := ADR(str);
pto := ADR(REPLACE_UML);
ptm := pto + INT_TO_DWORD(string_length);
pt1 := ADR(su);
pt2 := pt1 + 1;
L := LEN(str);
WHILE pos < L AND pos < string_length DO
	IF pt^ < 127 THEN
		(* no uml character simlply copy the character*)
		pto^ := pt^;
	ELSE
		(* convert the uml character *)
		su := TO_UML(pt^);
		(* we must make sure pointer are not out of range *)
		pto^ := pt1^;
		IF pto < ptm AND pt2^ > 0 THEN
			pto := pto + 1;
			pto^ := pt2^;
		END_IF;
	END_IF;
	(* increment pointers *)
	pt := pt + 1;
	pto := pto + 1;
	pos := pos + 1;
END_WHILE;

(* properly close the output string *)
pto^ := 0;

(* revision history
hm	29. feb 2008	rev 1.0
	original version

hm	29. mar. 2008	rev 1.1
	changed STRING to STRING(STRING_LENGTH)
	new code to avoid pointer out of range
	use new function to_uml
*)
END_FUNCTION

(* ---- RES_NI.st ---- *)
FUNCTION RES_NI : REAL
VAR_INPUT
    T : REAL;
    R0 : REAL;
END_VAR

VAR CONSTANT
    A : REAL := 0.5485;
    B : REAL := 0.000665;
    C : REAL := 2.805E-09;
END_VAR

VAR
    T2 : REAL;
END_VAR
T2 := T * T;
RES_NI := R0 + A * T + B * T2 + C * T2 * T2;

(* revision history

hm	4.8.2006		rev 1.0
	original version

hm	13.9.2007		rev 1.1
	changed coding for better performance

hm	2. dec. 2007	rev 1.2
	changed code for better performance
*)

(*

 Auszug aus DIN 43760 für Ni100

°C		R		°C		R		°C	R		°C		R		°C		R

-60 	69,5 	-10 	94,6 	40 	123,0 	90 		154,9 	140 	190,9
-55 	71,9 	-5 		97,3 	45 	126,0 	95 		158,3 	145 	194,8
-50 	74,3 	0 		100,0 	50 	129,1 	100 	161,8 	150 	198,7
-45 	76,7 	5 		102,8 	55 	132,2 	105 	165,3 	155 	202,6
-40 	79,1 	10 		105,6 	60 	135,3 	110 	168,8 	160 	206,6
-35 	81,6 	15 		108,4 	65 	138,5 	115 	172,4 	165 	210,7
-30 	84,2 	20 		111,2 	70 	141,7 	120 	176,0 	170 	214,8
-25 	86,7 	25 		114,1 	75 	145,0 	125 	179,6 	175 	219,0
-20 	89,3 	30 		117,1 	80 	148,3 	130 	183,3 	180 	223,2
-15 	91,9 	35 		120,0 	85 	151,6 	135 	187,1

*)
END_FUNCTION

(* ---- RES_NTC.st ---- *)
FUNCTION RES_NTC : REAL
VAR_INPUT
    T : REAL;
    RN : REAL;
    B : REAL;
END_VAR
RES_NTC := RN * EXP(B * (1.0 / (T+273.15) - 0.00335401643468053));

(* revision history

hm 30. dec. 2008	rev 1.0
	original version

hm	11. mar. 2009	rev 1.1
	changed real constants to use dot syntax

*)
END_FUNCTION

(* ---- RES_PT.st ---- *)
FUNCTION RES_PT : REAL
VAR_INPUT
    T : REAL;
    R0 : REAL;
END_VAR

VAR CONSTANT
    A : REAL := 0.00390802;
    B : REAL := -5.802E-07;
    C : REAL := -4.2735E-12;
END_VAR

VAR
    T2 : REAL;
END_VAR
T2 := T * T;

IF T >= 0.0 THEN
	RES_PT := R0 * ( 1.0 + A * T + B * T2);
ELSE
	RES_PT := R0 * ( 1.0 + A * T + B * T2 + C * (T - 100.0) * T2 * T);
END_IF;

(* revision history
hm	4. aug. 2006	rev 1.1
	original version

hm	2. dec 2007	rev 1.2
	changed code for better performance

hm	11. mar. 2009	rev 1.3
	changed real constants to use dot syntax

*)

(*
 Auszug aus DIN 43760 für Pt100

°C		R		°C		R		°C	R			°C		R			°C		R			°C		R

-200 	18,49 	-100 	60,25 	0 	100,00 	100 	138,50 	200 	175,84 	300 	212,02
-195 	20,65 	-95 	62,28 	5 	101,95 	105 	140,39 	205 	177,68 	305 	213,80
-190 	22,80 	-90 	64,30 	10 	103,90 	110 	142,29 	210 	179,51 	310 	215,57
-185 	24,94 	-85 	66,31 	15 	105,85 	115 	144,17 	215 	181,34 	315 	217,35
-180 	27,08 	-80 	68,33 	20 	107,79 	120 	146,06 	220 	183,17 	320 	219,12
-175 	29,20 	-75 	70,33 	25 	109,73 	125 	147,94 	225 	184,99 	325 	220,88
-170 	31,32 	-70 	72,33 	30 	111,67 	130 	149,82 	230 	186,82 	330 	222,65
-165 	33,43 	-65 	74,33 	35 	113,61 	135 	151,70 	235 	188,63 	335 	224,41
-160 	35,33 	-60 	76,33 	40 	115,54 	140 	153,58 	240 	190,45 	340 	226,17
-155 	37,63 	-55 	78,32 	45 	117,47 	145 	155,45 	245 	192,26 	345 	227,92
-150 	39,71 	-50 	80,31 	50 	119,40 	150 	157,31 	250 	194,07 	350 	229,67
-145 	41,79 	-45 	82,29 	55 	121,32 	155 	159,18 	255 	195,88 	355 	231,42
-140 	43,87 	-40 	84,27 	60 	123,24 	160 	161,04 	260 	197,69 	360 	233,17
-135 	45,94 	-35 	86,25 	65 	125,16 	165 	162,90 	265 	199,49 	365 	234,91
-130 	48,00 	-30 	88,22 	70 	127,07 	170 	164,76 	270 	201,29 	370 	236,65
-125 	50,06 	-25 	90,19 	75 	128,98 	175 	166,61 	275 	203,08 	375 	238,39
-120 	52,11 	-20 	92,16 	80 	130,89 	180 	168,46 	280 	204,88 	380 	240,13
-115 	54,15 	-15 	94,12 	85 	132,80 	185 	170,31 	285 	206,67 	385 	241,86
-110 	56,19 	-10 	96,09 	90 	134,70 	190 	172,16 	290 	208,45 	390 	243,59
-105 	58,22 	-5 		98,04 	95 	136,60 	195 	174,00 	295 	210,24 	395 	245,31

*)
(*
revision history

*)
END_FUNCTION

(* ---- RES_SI.st ---- *)
FUNCTION RES_SI : REAL
VAR_INPUT
    T : REAL;
    RS : REAL;
    TS : REAL;
END_VAR

VAR_CONSTANT
    A : REAL := 0.00764;
    B : REAL := 1.66E-05;
END_VAR

VAR
    TX : REAL;
END_VAR
TX := T - TS;
RES_SI := RS * ( 1.0 + A * TX + B * TX * TX);

(* revision history
hm	4. aug 2006	rev 1.0
	original version

hm	2. dec 2007	rev 1.1
	changed code for better performance

hm	11. mar. 2009	rev 1.2
	changed real constants to use dot syntax

*)
END_FUNCTION

(* ---- REVERSE.st ---- *)
FUNCTION REVERSE : BYTE
VAR_INPUT
    IN : BYTE;
END_VAR
(* new code donated by rebler wolfgang *)
REVERSE := ROR(in,1) AND 2#10001000 OR ROL(in,1) AND 2#00010001 OR ROR(in,3) AND 2#01000100 OR ROL(in,3) AND 2#00100010;

(* old code
REVERSE := SHL(in,7) OR SHR(in,7) OR (ROR(in,3) AND 2#01000100) OR (ROL(in,3) AND 2#00100010)
	OR (SHL(in,1) AND 2#00010000) OR (SHR(in,1) AND 2#00001000);
*)

(* revision history
hm		9.oct 2007		rev 1.0
	original version

hm		18. feb 2008	rev 1.1
	improved performance

RW    3. feb. 2021  	rev 1.2
	improved performance
*)
END_FUNCTION

(* ---- RND.st ---- *)
FUNCTION RND : REAL
VAR_INPUT
    X : REAL;
    N : INT;
END_VAR_INPUT

VAR
    M : REAL;
END_VAR
IF X = 0.0 THEN
	RND := 0.0;
ELSE
	M := EXPN(10.0,N - CEIL(LOG(ABS(X))));
	RND := DINT_TO_REAL(REAL_TO_DINT(X * M)) / M;
END_IF;

(* revision history
hm	11. mar 2008	rev 1.0
	original version

hm	26. oct. 2008	rev 1.1
	code optimization

hm	10. mar. 2009	rev 1.2
	real constants updated to new systax using dot

*)
END_FUNCTION

(* ---- ROUND.st ---- *)
FUNCTION ROUND : REAL
VAR_INPUT
    in : REAL;
    N : INT;
END_VAR

VAR
    X : REAL;
END_VAR
X := setup.DECADES[LIMIT(0,N,8)];
ROUND := DINT_TO_REAL(REAL_TO_DINT(in * X)) / X;

(* revision history
hm	1. sep 2006	rev 1.0
	original version

hm	2. dec 2007	rev 1.1
	changed code for better performance

hm	8. jan 2008	rev 1.2
	further improvement in performance

hm 11. mar. 2008	rev 1.3
	corrected an error with negative numbers
	use real_to_dint instead of trunc

hm	16. mar 2008	rev 1.4
	added type conversion to avoid warning under codesys 3.0

hm	25. oct. 2008	rev 1.5
	new code using global constants decades
*)
END_FUNCTION

(* ---- SCALE.st ---- *)
FUNCTION SCALE : REAL
VAR_INPUT
    X : REAL;
    K : REAL;
    O : REAL;
    MX : REAL;
    MN : REAL;
END_VAR
SCALE := LIMIT(MN, X * K + O, MX);

(* revision history
hm	16. may. 2008		rev 1.0
	original version
*)
END_FUNCTION

(* ---- SCALE_B.st ---- *)
FUNCTION SCALE_B : REAL
VAR_INPUT
    X: BYTE;
    I_LO: BYTE;
    I_HI: BYTE;
    O_LO: REAL;
    O_HI: REAL;
END_VAR
IF I_HI = I_LO THEN
	SCALE_B := O_LO;
ELSE
	SCALE_B := (O_HI - O_LO) / BYTE_TO_REAL(I_HI - I_LO) * BYTE_TO_REAL(LIMIT(I_LO, X, I_HI));
END_IF

(* revision history
hm	18. may. 2008		rev 1.0
	original version

hm	18. jan 2011		rev 1.1
	avoid division by 0

*)
END_FUNCTION

(* ---- SCALE_B2.st ---- *)
FUNCTION SCALE_B2 : REAL
VAR_INPUT
    in1 : BYTE;
    in2 : BYTE;
    K : REAL;
    O : REAL;
    in1_min : REAL; // input_constant
    in1_max : REAL := 1000.0; // input_constant
    in2_min : REAL; // input_constant
    in2_max : REAL := 1000.0; // input_constant
END_VAR
SCALE_B2 := 	(((in1_max - in1_min)* in1 + (in2_max - in2_min)* in2) * 0.003921569 + in1_min + in2_min) * K + O;

(* revision History
hm 19.1.2007		rev 1.1
	changed outputs to real to avoid overflow of integer
	added offset for better cascading of scale functions
	changed from FB to function

hm	6. jan 2008		rev 1.2
	improved performance

hm	26. oct. 2008	rev 1.3
	code optimization

hm	3. nov. 2008	rev 1.4
	used wrong factor in formula

*)
END_FUNCTION

(* ---- SCALE_B4.st ---- *)
FUNCTION SCALE_B4 : REAL
VAR_INPUT
    in1 : BYTE;
    in2 : BYTE;
    in3 : BYTE;
    in4 : BYTE;
    K : REAL;
    O : REAL;
    in1_min : REAL;
    in1_max : REAL := 1000.0;
    in2_min : REAL;
    in2_max : REAL := 1000.0;
    in3_min : REAL;
    in3_max : REAL := 1000.0;
    in4_min : REAL;
    in4_max : REAL := 1000.0;
END_VAR
SCALE_B4 := 	(((in1_max - in1_min)* in1 + (in2_max - in2_min)* in2 + (in3_max - in3_min)* in3 + (in4_max - in4_min)* in4)* 0.003921569 + in1_min + in2_min + in3_min + in4_min) * K + O;

(* revision History
hm 19.1.2007		rev 1.1
	changed outputs to real to avoid overflow of integer
	added offset for better cascading of scale functions
	changed from fb to function

hm	6. jan 2008		rev 1.2
	improved performance

hm	26. oct. 2008	rev 1.3
	optimized code

hm	3. nov. 2008	rev 1.4
	used wrong factor in formula

*)
END_FUNCTION

(* ---- SCALE_B8.st ---- *)
FUNCTION SCALE_B8 : REAL
VAR_INPUT
    in1 : BYTE;
    in2 : BYTE;
    in3 : BYTE;
    in4 : BYTE;
    in5 : BYTE;
    in6 : BYTE;
    in7 : BYTE;
    in8 : BYTE;
    K : REAL;
    O : REAL;
    in1_min : REAL;
    in1_max : REAL := 1000.0;
    in2_min : REAL;
    in2_max : REAL := 1000.0;
    in3_min : REAL;
    in3_max : REAL := 1000.0;
    in4_min : REAL;
    in4_max : REAL := 1000.0;
    in5_min : REAL;
    in5_max : REAL := 1000.0;
    in6_min : REAL;
    in6_max : REAL := 1000.0;
    in7_min : REAL;
    in7_max : REAL := 1000.0;
    in8_min : REAL;
    in8_max : REAL := 1000.0;
END_VAR
SCALE_B8 := 	(((in1_max - in1_min)* in1 + (in2_max - in2_min)* in2 + (in3_max - in3_min)* in3 + (in4_max - in4_min)* in4 +
				(in5_max - in5_min)* in5 + (in6_max - in6_min)* in6 + (in7_max - in7_min)* in7 + (in8_max - in8_min)* in8) * 0.003921569
				 + in1_min + in2_min + in3_min + in4_min + in5_min + in6_min + in7_min + in8_min) * K + O;

(* revision History
hm	19. jan.2007	rev 1.1
	changed outputs to real to avoid overflow of integer
	added offset for better cascading of scale functions

hm	6. jan. 2008	rev 1.2
	improved performance

hm	26. oct. 2008	rev 1.3
	code optimization

hm	3. nov. 2008	rev 1.4
	used wrong factor in formula

*)
END_FUNCTION

(* ---- SCALE_D.st ---- *)
FUNCTION SCALE_D : REAL
VAR_INPUT
    X : DWORD;
    I_LO : DWORD;
    I_HI : DWORD;
    O_LO : REAL;
    O_HI : REAL;
END_VAR
IF I_HI = I_LO THEN
	SCALE_D := O_LO;
ELSE
	SCALE_D := (O_HI - O_LO) / DWORD_TO_REAL(I_HI - I_LO) * DWORD_TO_REAL(LIMIT(I_LO, X, I_HI) - I_LO) + O_LO;
END_IF;

(* revision history
hm	18. may. 2008	rev 1.0
	original version

hm	13. nov. 2008	rev 1.1
	corrected formula for negative gradient

hm	11. jan 2011	rev 1.2
	avoid division by 0
*)
END_FUNCTION

(* ---- SCALE_R.st ---- *)
FUNCTION SCALE_R : REAL
VAR_INPUT
    X    : REAL;
    I_LO : REAL;
    I_HI : REAL;
    O_LO : REAL;
    O_HI : REAL;
END_VAR
IF I_LO = I_HI THEN
	SCALE_R := O_LO;
ELSE
	SCALE_R := (O_HI - O_LO) / (I_HI - I_LO) * (LIMIT(I_LO, X, I_HI) - I_LO) + O_LO;
END_IF;

(* revision history
hm	18. may. 2008	rev 1.0
	original version

hm	13. nov. 2008	rev 1.1
	corrected formula for negative gradient

hm	11. jan 2011	rev 1.2
	avoid division by 0

*)
END_FUNCTION

(* ---- SCALE_X2.st ---- *)
FUNCTION SCALE_X2 : REAL
VAR_INPUT
    IN1 : BOOL;
    IN2 : BOOL;
    K : REAL;
    O : REAL;
    IN1_MIN : REAL;
    IN1_MAX : REAL := 1000.0;
    IN2_MIN : REAL;
    IN2_MAX : REAL := 1000.0;
END_VAR
SCALE_X2 := (SEL(IN1, IN1_MIN, IN1_MAX)+ SEL(IN2, IN2_MIN, IN2_MAX)) * k + o;

(* revision history
hm	19. jan, 2007	rev 1.0
	original version

hm	26. oct. 2008	rev 1.1
	code optimized

*)
END_FUNCTION

(* ---- SCALE_X4.st ---- *)
FUNCTION SCALE_X4 : REAL
VAR_INPUT
    IN1 : BOOL;
    IN2 : BOOL;
    IN3 : BOOL;
    IN4 : BOOL;
    K : REAL;
    O : REAL;
    IN1_MIN : REAL; // input_constant
    IN1_MAX : REAL := 1000.0; // input_constant
    IN2_MIN : REAL; // input_constant
    IN2_MAX : REAL := 1000.0; // input_constant
    IN3_MIN : REAL; // input_constant
    IN3_MAX : REAL := 1000.0; // input_constant
    IN4_MIN : REAL; // input_constant
    IN4_MAX : REAL := 1000.0; // input_constant
END_VAR
SCALE_X4 := (SEL(IN1,IN1_MIN, IN1_MAX) + SEL(IN2, IN2_MIN, IN2_MAX)+SEL(IN3, IN3_MIN, IN3_MAX)+ SEL(IN4, IN4_MIN, IN4_MAX)) * k + o;

(* revision history
hm	19. jan. 2008	rev 1.0
	original version

hm	26. oct. 2008	rev 1.1
	optimized code
*)
END_FUNCTION

(* ---- SCALE_X8.st ---- *)
FUNCTION SCALE_X8 : REAL
VAR_INPUT
    in1 : BOOL;
    in2 : BOOL;
    in3 : BOOL;
    in4 : BOOL;
    in5 : BOOL;
    in6 : BOOL;
    in7 : BOOL;
    in8 : BOOL;
    K : REAL;
    O : REAL;
    in1_min : REAL; // input_constant
    in1_max : REAL := 1000.0; // input_constant
    in2_min : REAL; // input_constant
    in2_max : REAL := 1000.0; // input_constant
    in3_min : REAL; // input_constant
    in3_max : REAL := 1000.0; // input_constant
    in4_min : REAL; // input_constant
    in4_max : REAL := 1000.0; // input_constant
    in5_min : REAL; // input_constant
    in5_max : REAL := 1000.0; // input_constant
    in6_min : REAL; // input_constant
    in6_max : REAL := 1000.0; // input_constant
    in7_min : REAL; // input_constant
    in7_max : REAL := 1000.0; // input_constant
    in8_min : REAL; // input_constant
    in8_max : REAL := 1000.0; // input_constant
END_VAR
SCALE_X8 := (SEL(IN1,IN1_MIN, IN1_MAX)+ SEL(IN2,IN2_MIN, IN2_MAX)+SEL(IN3,IN3_MIN, IN3_MAX)+ SEL(IN4,IN4_MIN, IN4_MAX)
				+SEL(IN5,IN5_MIN, IN5_MAX)+ SEL(IN6,IN6_MIN, IN6_MAX)+SEL(IN7,IN7_MIN, IN7_MAX)+ SEL(IN8,IN8_MIN, IN8_MAX)) * k + o;

(* revision history
hm	19. jan. 2008	rev 1.0
	original version

hm	26. oct. 2008	rev 1.1
	optimized code

hm	24. jan. 2008	rev 1.2
	corrected error in formula
*)
END_FUNCTION

(* ---- SDT_TO_DATE.st ---- *)
FUNCTION SDT_TO_DATE : DATE
VAR_INPUT
    DTI : SDT;
END_VAR
SDT_TO_DATE := SET_DATE(DTI.YEAR, DTI.MONTH, DTI.DAY);

(* revision history

hm 18. oct. 2008	rev 1.0
	original version

*)
END_FUNCTION

(* ---- SDT_TO_DT.st ---- *)
FUNCTION SDT_TO_DT : DT
VAR_INPUT
    DTI : SDT;
END_VAR
SDT_TO_DT := SET_DT(DTI.YEAR, DTI.MONTH, DTI.DAY, DTI.HOUR, DTI.MINUTE, DTI.SECOND);

(* revision history

hm 18. oct. 2008	rev 1.0
	original version

*)
END_FUNCTION

(* ---- SDT_TO_TOD.st ---- *)
FUNCTION SDT_TO_TOD : TOD
VAR_INPUT
    DTI: SDT; // Derived data type
END_VAR
SDT_TO_TOD := DWORD_TO_TOD(INT_TO_DWORD(DTI.HOUR) * 3600000 + INT_TO_DWORD(DTI.MINUTE) * 60000 + INT_TO_DWORD(DTI.SECOND) * 1000 + INT_TO_DWORD(DTI.MS));

(* revision history

hm 18. oct. 2008	rev 1.0
	original version

hm	16. nov. 2008	rev 1.1
	added typecasts to avoid warnings
*)
END_FUNCTION

(* ---- SECOND.st ---- *)
FUNCTION SECOND : REAL
VAR_INPUT
    itod : TOD;
END_VAR
SECOND := DWORD_TO_REAL(TOD_TO_DWORD(itod) - TOD_TO_DWORD(itod)/60000 * 60000) / 1000.0;

(* change history

hm	2. oct. 2006 rev 1.1
	changed name of input to itod

*)
END_FUNCTION

(* ---- SECOND_OF_DT.st ---- *)
FUNCTION SECOND_OF_DT : INT
VAR_INPUT
    XDT : DT;
END_VAR
SECOND_OF_DT := DWORD_TO_INT(DT_TO_DWORD(XDT) MOD 60);

(* revision history
hm		6.9.2008	rev 1.0
	original version

*)
END_FUNCTION

(* ---- SECOND_TO_TIME.st ---- *)
FUNCTION SECOND_TO_TIME : TIME
VAR_INPUT
    IN : REAL;
END_VAR
SECOND_TO_TIME := DWORD_TO_TIME(REAL_TO_DWORD(IN * 1000.0));

(* revision history
hm	4. aug. 2006	rev 1.0
	original version

hm	14. mar. 2008	rev 1.1
	rounded the input after the last digit

hm	24. feb. 2009	rev 1.2
	changed input to IN
*)
END_FUNCTION

(* ---- SENSOR_INT.st ---- *)
FUNCTION SENSOR_INT : REAL
VAR_INPUT
    Voltage : REAL;
    Current : REAL;
    RP : REAL;
    RS : REAL;
END_VAR

VAR
    RG : REAL;
END_VAR
IF current <> 0.0 THEN
	RG := voltage / current;
	SENSOR_INT := RP * ( RG - RS) / ( RP + RS - RG);
END_IF;

(* revisaion history

hm 20.1.2007		rev 1.1
	deleted input R0 which was not needed.

hm	2. dec 2007	rev 1.2
	corrected an error in formula and improoved speed

hm	11. mar. 2009	rev 1.3
	changed real constants to use dot syntax

*)
END_FUNCTION

(* ---- SET_DATE.st ---- *)
FUNCTION SET_DATE : DATE
VAR_INPUT
    YEAR : INT;
    MONTH : INT;
    DAY : INT;
END_VAR_INPUT

VAR
    count : INT;
    ofs : ARRAY[1..12] OF INT := [0, 31, 59, 90, 120, 151, 181, 212, 243, 273, 304, 334];
    ENDIF : BOOL;
END_VAR
IF (MONTH > 2) AND (SHL(YEAR,14) = 0)
THEN (* we add one day for leap year *)
	SET_DATE := DWORD_TO_DATE((INT_TO_DWORD(ofs[MONTH] + day ) + SHR(INT_TO_DWORD(year) * 1461 - 2878169, 2))*86400);
ELSE
	SET_DATE := DWORD_TO_DATE((INT_TO_DWORD(ofs[MONTH] + day - 1 ) + SHR(INT_TO_DWORD(year) * 1461 - 2878169, 2))*86400);
END_IF;

(* old code
IF month > 2 THEN
	count := (month - 1) * 30;
	IF month > 7 THEN count := count + SHR(month - 3,1); ELSE count := count + SHR(month - 4,1); END_IF;
	(* chech for leap year and add one day if true *)
	IF SHL(year,14) = 0 THEN count := count + 1; END_IF;
ELSE
	count := (month - 1) * 31;
END_IF;

SET_DATE := DWORD_TO_DATE((INT_TO_DWORD(count + day - 1) + SHR(INT_TO_DWORD(year) * 1461 - 2878169, 2)) * 86400);
*)

(* revision history
hm	4. aug. 2006	rev 1.0
	original version

hm	19 sep. 2007	rev 1.1
	use function leap_year to calculate leap year, more exceptions are handled

hm	1. okt	2007	rev 1.2
	added compatibility to step7

hm	16.dec 2007		rev 1.3
	changed code to improove performance

hm	3. jan. 2008	rev 1.4
	further improvements in performance

hm	16. mar. 2008	rev 1.5
	added type conversions to avoid warnings under codesys 3.0

hm	7. apr. 2008	rev 1.6
	deleted unused step7 code

hm	14. oct. 2008	rev 1.7
	optimized code for better performance

hm	25. oct. 2008	rev 2.0
	new code using setup constants

hm	16. nov. 2008	rev 2.1
	added typecasts to avoid warnings

hm	22. jan. 2011	rev 2.2
	improved performance

hm	29. dec. 2011	rev 2.3
	improved performance

hm 3. FEB 2021 rev 2.4
	new code to be more readable
*)
END_FUNCTION

(* ---- SET_DT.st ---- *)
FUNCTION SET_DT : DT
VAR_INPUT
    year : INT;
    month : INT;
    day : INT;
    hour : INT;
    minute : INT;
    second : INT;
END_VAR
SET_DT := DWORD_TO_DT(DATE_TO_DWORD(SET_DATE(YEAR, MONTH, day)) + INT_TO_DWORD(SECOND) + INT_TO_DWORD(MINUTE) * 60 + INT_TO_DWORD(HOUR) * 3600);

(* revision history
hm	4. aug. 2006		rev 1.0
	original version

hm		19 sep. 2007	rev 1.1
	use function leap_year to calculate leap year, more exceptions are handled

hm		1. okt 2007		rev 1.2
	added step7 compatibility
	call function set_date

hm		8. oct 2007		rev 1.3
	deleted unused variables count and leap

hm		1. 11 2007		rev 1.4
	converted hour type integer to dword in calculation to avoid overrun on möller ecp4

hm		16. mar 2008	rev 1.5
	added type conversions to avoid warnings under codesys 3.0
*)
END_FUNCTION

(* ---- SET_TOD.st ---- *)
FUNCTION SET_TOD : TOD
VAR_INPUT
    hour : INT;
    minute : INT;
    second : REAL;
END_VAR
SET_TOD := DWORD_TO_TOD(REAL_TO_DWORD(SECOND * 1000.0) + INT_TO_DWORD(MINUTE) * 60000 + INT_TO_DWORD(HOUR) * 3600000);

(* revision history

hm		4.aug.2006		rev 1.0
	original version

hm		11. sep 2007	rev 1.1
	changed coding to avoid a compiler warning under twincat.

hm		1. nov 2007	rev 1.2
	changed coding to avoid possible overrun situation on möller ecp4

hm		2. Nov	2007	rev 1.3
	changed dword to DINT in calcualtion to avoid warnings with some compilers

hm		14. mar 2008	rev 1.4
	changed code to avoid rounding problem at last digit of millisecond

hm		16. mar. 2008	rev 1.5
	added type conversions to avoid warning under codesys 3.0
*)
END_FUNCTION

(* ---- SGN.st ---- *)
FUNCTION SGN : INT
VAR_INPUT
    X : REAL;
END_VAR
IF X > 0 THEN
	SGN := 1;
ELSIF X < 0 THEN
	SGN := -1;
ELSE
	SGN := 0;
END_IF;

(* revision histroy
hm	16. oct 2007	rev 1.0
	original version

hm	11. nov 2007	rev 1.1
	changed type of function from real to int

*)
END_FUNCTION

(* ---- SHL1.st ---- *)
FUNCTION SHL1 : DWORD
VAR_INPUT
    IN : DWORD;
    N : INT;
END_VAR

VAR_CONSTANT
    temp : DWORD := 16#FFFFFFFF;
END_VAR
SHL1 := SHR(temp,32-N) OR SHL(IN,N);

(* revision history
hm	14.9.2007		rev 1.0
	original version

hm	27. dec 2007	rev 1.1
	changed code for better performance

*)
END_FUNCTION

(* ---- SHR1.st ---- *)
FUNCTION SHR1 : DWORD
VAR_INPUT
    IN : DWORD;
    N : INT;
END_VAR

VAR_CONSTANT
    temp : DWORD := 16#FFFFFFFF;
END_VAR
SHR1 := SHL(temp,32-N) OR SHR(IN,N);

(* revision history
hm	14.9.2007		rev 1.0
	original version

hm	27. dec 2007	rev 1.1
	changed code for better performance

*)
END_FUNCTION

(* ---- SIGMOID.st ---- *)
FUNCTION SIGMOID : REAL
VAR_INPUT
    X : REAL;
END_VAR
IF X > 20.0 THEN
	SIGMOID := 1.0;
ELSIF x < -85.0 THEN
	SIGMOID := 0.0;
ELSE
	SIGMOID := 1.0 / (1.0 + EXP(-X));
END_IF;

(* revision history
hm	10.12.2007		rev 1.0
	original version

hm	11. mar. 2008		rev 1.1
	extended range of valid inputs to +inv / -inv

hm 10. mar. 2009		rev 1.2
	real constants updated to new systax using dot

*)
END_FUNCTION
